LIN {X 0,Y 474.607,Z 153.704,A -85,B 0,C 180,E1 -7123.223,E2 -7123.223} C_VEL
LIN {X 0,Y 474.574,Z 152.961,A -85,B 0,C 180,E1 -7123.313,E2 -7123.313} C_VEL
LIN {X 0,Y 474.891,Z 139.856,A -85,B 0,C 180,E1 -7126.331,E2 -7126.331} C_VEL
LIN {X 0,Y 475.169,Z 128.62,A -85,B 0,C 180,E1 -7128.989,E2 -7128.989} C_VEL
LIN {X 0,Y 474.717,Z 124.266,A -85,B 0,C 180,E1 -7130.105,E2 -7130.105} C_VEL
LIN {X 0,Y 474.611,Z 124.173,A -85,B 0,C 180,E1 -7133.566,E2 -7133.566} C_VEL
LIN {X 0,Y 474.655,Z 124.176,A -85,B 0,C 180,E1 -7136.372,E2 -7136.372} C_VEL
LIN {X 0,Y 474.621,Z 124.172,A -85,B 0,C 180,E1 -7139.252,E2 -7139.252} C_VEL
LIN {X 0,Y 474.614,Z 124.178,A -85,B 0,C 180,E1 -7142.43,E2 -7142.43} C_VEL
LIN {X 0,Y 474.617,Z 124.174,A -85,B 0,C 180,E1 -7145.469,E2 -7145.469} C_VEL
LIN {X 0,Y 474.611,Z 124.175,A -85,B 0,C 180,E1 -7148.457,E2 -7148.457} C_VEL
LIN {X 0,Y 474.627,Z 124.172,A -85,B 0,C 180,E1 -7150.959,E2 -7150.959} C_VEL
LIN {X 0,Y 474.605,Z 124.177,A -85,B 0,C 180,E1 -7154.105,E2 -7154.105} C_VEL
LIN {X 0,Y 474.613,Z 124.175,A -85,B 0,C 180,E1 -7157.065,E2 -7157.065} C_VEL
LIN {X 0,Y 474.617,Z 124.173,A -85,B 0,C 180,E1 -7160.354,E2 -7160.354} C_VEL
LIN {X 0,Y 474.591,Z 124.18,A -85,B 0,C 180,E1 -7163.677,E2 -7163.677} C_VEL
LIN {X 0,Y 474.642,Z 124.172,A -85,B 0,C 180,E1 -7166.78,E2 -7166.78} C_VEL
LIN {X 0,Y 474.604,Z 124.175,A -85,B 0,C 180,E1 -7169.77,E2 -7169.77} C_VEL
LIN {X 0,Y 474.696,Z 124.167,A -85,B 0,C 180,E1 -7172.68,E2 -7172.68} C_VEL
LIN {X 0,Y 474.656,Z 124.169,A -85,B 0,C 180,E1 -7175.507,E2 -7175.507} C_VEL
LIN {X 0,Y 474.67,Z 124.169,A -85,B 0,C 180,E1 -7179.185,E2 -7179.185} C_VEL
LIN {X 0,Y 474.656,Z 124.168,A -85,B 0,C 180,E1 -7181.884,E2 -7181.884} C_VEL
LIN {X 0,Y 474.699,Z 124.171,A -85,B 0,C 180,E1 -7184.544,E2 -7184.544} C_VEL
LIN {X 0,Y 474.738,Z 124.161,A -85,B 0,C 180,E1 -7188.038,E2 -7188.038} C_VEL
LIN {X 0,Y 474.727,Z 124.159,A -85,B 0,C 180,E1 -7191.486,E2 -7191.486} C_VEL
LIN {X 0,Y 474.778,Z 124.159,A -85,B 0,C 180,E1 -7194.052,E2 -7194.052} C_VEL
LIN {X 0,Y 474.893,Z 124.14,A -85,B 0,C 180,E1 -7197.455,E2 -7197.455} C_VEL
LIN {X 0,Y 474.911,Z 124.144,A -85,B 0,C 180,E1 -7200,E2 -7200} C_VEL
LIN {X 0,Y 474.893,Z 124.139,A -85,B 0,C 180,E1 -7202.545,E2 -7202.545} C_VEL
LIN {X 0,Y 474.777,Z 124.158,A -85,B 0,C 180,E1 -7205.948,E2 -7205.948} C_VEL
LIN {X 0,Y 474.726,Z 124.159,A -85,B 0,C 180,E1 -7208.513,E2 -7208.513} C_VEL
LIN {X 0,Y 474.703,Z 124.165,A -85,B 0,C 180,E1 -7211.962,E2 -7211.962} C_VEL
LIN {X 0,Y 474.698,Z 124.17,A -85,B 0,C 180,E1 -7215.456,E2 -7215.456} C_VEL
LIN {X 0,Y 474.664,Z 124.172,A -85,B 0,C 180,E1 -7219.01,E2 -7219.01} C_VEL
LIN {X 0,Y 474.586,Z 124.178,A -85,B 0,C 180,E1 -7221.729,E2 -7221.729} C_VEL
LIN {X 0,Y 474.655,Z 124.17,A -85,B 0,C 180,E1 -7224.493,E2 -7224.493} C_VEL
LIN {X 0,Y 474.679,Z 124.168,A -85,B 0,C 180,E1 -7227.334,E2 -7227.334} C_VEL
LIN {X 0,Y 474.603,Z 124.176,A -85,B 0,C 180,E1 -7230.23,E2 -7230.23} C_VEL
LIN {X 0,Y 474.641,Z 124.172,A -85,B 0,C 180,E1 -7233.22,E2 -7233.22} C_VEL
LIN {X 0,Y 474.59,Z 124.181,A -85,B 0,C 180,E1 -7236.323,E2 -7236.323} C_VEL
LIN {X 0,Y 474.616,Z 124.173,A -85,B 0,C 180,E1 -7239.646,E2 -7239.646} C_VEL
LIN {X 0,Y 474.613,Z 124.175,A -85,B 0,C 180,E1 -7242.934,E2 -7242.934} C_VEL
LIN {X 0,Y 474.604,Z 124.178,A -85,B 0,C 180,E1 -7245.895,E2 -7245.895} C_VEL
LIN {X 0,Y 474.626,Z 124.172,A -85,B 0,C 180,E1 -7249.041,E2 -7249.041} C_VEL
LIN {X 0,Y 474.609,Z 124.178,A -85,B 0,C 180,E1 -7251.704,E2 -7251.704} C_VEL
LIN {X 0,Y 474.626,Z 124.172,A -85,B 0,C 180,E1 -7254.726,E2 -7254.726} C_VEL
LIN {X 0,Y 474.634,Z 124.179,A -85,B 0,C 180,E1 -7257.788,E2 -7257.788} C_VEL
LIN {X 0,Y 474.623,Z 124.173,A -85,B 0,C 180,E1 -7260.885,E2 -7260.885} C_VEL
LIN {X 0,Y 474.661,Z 124.175,A -85,B 0,C 180,E1 -7263.629,E2 -7263.629} C_VEL
LIN {X 0,Y 474.635,Z 124.143,A -85,B 0,C 180,E1 -7266.642,E2 -7266.642} C_VEL
LIN {X 0,Y 474.654,Z 124.24,A -85,B 0,C 180,E1 -7267.156,E2 -7267.156} C_VEL
LIN {X 0,Y 475.653,Z 130.342,A -85,B 0,C 180,E1 -7268.568,E2 -7268.568} C_VEL
LIN {X 0,Y 475.455,Z 140.784,A -85,B 0,C 180,E1 -7270.799,E2 -7270.799} C_VEL
LIN {X 0,Y 474.832,Z 156.822,A -85,B 0,C 180,E1 -7274.168,E2 -7274.168} C_VEL
LIN {X 0,Y 474.475,Z 169.531,A -85,B 0,C 180,E1 -7276.78,E2 -7276.78} C_VEL
LIN {X 0,Y 474.997,Z 173.212,A -85,B 0,C 180,E1 -7276.9,E2 -7276.9} C_VEL
LIN {X 0,Y 476.416,Z 185.772,A -85,B 0,C 180,E1 -7277.13,E2 -7277.13} C_VEL
LIN {X 0,Y 476.155,Z 245.998,A -85,B 0,C 180,E1 -7278.055,E2 -7278.055} C_VEL
LIN {X 0,Y 475.911,Z 254.89,A -85,B 0,C 180,E1 -7278.285,E2 -7278.285} C_VEL
LIN {X 0,Y 475.705,Z 264.57,A -85,B 0,C 180,E1 -7278.658,E2 -7278.658} C_VEL
LIN {X 0,Y 475.452,Z 273.742,A -85,B 0,C 180,E1 -7279.137,E2 -7279.137} C_VEL
LIN {X 0,Y 475.067,Z 284.557,A -85,B 0,C 180,E1 -7279.882,E2 -7279.882} C_VEL
LIN {X 0,Y 474.683,Z 293.871,A -85,B 0,C 180,E1 -7280.735,E2 -7280.735} C_VEL
LIN {X 0,Y 474.468,Z 300.546,A -85,B 0,C 180,E1 -7281.482,E2 -7281.482} C_VEL
LIN {X 0,Y 474.248,Z 306.882,A -85,B 0,C 180,E1 -7282.336,E2 -7282.336} C_VEL
LIN {X 0,Y 474.068,Z 312.147,A -85,B 0,C 180,E1 -7283.189,E2 -7283.189} C_VEL
LIN {X 0,Y 473.99,Z 316.538,A -85,B 0,C 180,E1 -7284.043,E2 -7284.043} C_VEL
LIN {X 0,Y 473.795,Z 321.713,A -85,B 0,C 180,E1 -7285.321,E2 -7285.321} C_VEL
LIN {X 0,Y 473.826,Z 325.514,A -85,B 0,C 180,E1 -7286.599,E2 -7286.599} C_VEL
LIN {X 0,Y 473.727,Z 327.26,A -85,B 0,C 180,E1 -7287.449,E2 -7287.449} C_VEL
LIN {X 0,Y 473.693,Z 328.512,A -85,B 0,C 180,E1 -7288.3,E2 -7288.3} C_VEL
LIN {X 0,Y 473.686,Z 329.292,A -85,B 0,C 180,E1 -7289.15,E2 -7289.15} C_VEL
LIN {X 0,Y 473.668,Z 329.587,A -85,B 0,C 180,E1 -7290,E2 -7290} C_VEL
LIN {X 0,Y 473.686,Z 329.291,A -85,B 0,C 180,E1 -7290.85,E2 -7290.85} C_VEL
LIN {X 0,Y 473.693,Z 328.509,A -85,B 0,C 180,E1 -7291.701,E2 -7291.701} C_VEL
LIN {X 0,Y 473.727,Z 327.256,A -85,B 0,C 180,E1 -7292.551,E2 -7292.551} C_VEL
LIN {X 0,Y 473.82,Z 324.353,A -85,B 0,C 180,E1 -7293.827,E2 -7293.827} C_VEL
LIN {X 0,Y 473.795,Z 321.706,A -85,B 0,C 180,E1 -7294.68,E2 -7294.68} C_VEL
LIN {X 0,Y 473.987,Z 316.527,A -85,B 0,C 180,E1 -7295.958,E2 -7295.958} C_VEL
LIN {X 0,Y 474.123,Z 309.701,A -85,B 0,C 180,E1 -7297.239,E2 -7297.239} C_VEL
LIN {X 0,Y 474.398,Z 302.239,A -85,B 0,C 180,E1 -7298.305,E2 -7298.305} C_VEL
LIN {X 0,Y 474.668,Z 294.88,A -85,B 0,C 180,E1 -7299.159,E2 -7299.159} C_VEL
LIN {X 0,Y 474.993,Z 287.001,A -85,B 0,C 180,E1 -7299.905,E2 -7299.905} C_VEL
LIN {X 0,Y 475.285,Z 278.674,A -85,B 0,C 180,E1 -7300.544,E2 -7300.544} C_VEL
LIN {X 0,Y 475.615,Z 268.044,A -85,B 0,C 180,E1 -7301.183,E2 -7301.183} C_VEL
LIN {X 0,Y 475.856,Z 256.486,A -85,B 0,C 180,E1 -7301.663,E2 -7301.663} C_VEL
LIN {X 0,Y 476.109,Z 246.824,A -85,B 0,C 180,E1 -7301.927,E2 -7301.927} C_VEL
LIN {X 0,Y 476.329,Z 197.947,A -85,B 0,C 180,E1 -7302.686,E2 -7302.686} C_VEL
LIN {X 0,Y 476.185,Z 182.261,A -85,B 0,C 180,E1 -7302.928,E2 -7302.928} C_VEL
LIN {X 0,Y 474.503,Z 169.838,A -85,B 0,C 180,E1 -7303.189,E2 -7303.189} C_VEL
LIN {X 0,Y 474.633,Z 164.918,A -85,B 0,C 180,E1 -7304.142,E2 -7304.142} C_VEL
LIN {X 0,Y 475.093,Z 149.174,A -85,B 0,C 180,E1 -7307.431,E2 -7307.431} C_VEL
LIN {X 0,Y 475.598,Z 135.504,A -85,B 0,C 180,E1 -7310.32,E2 -7310.32} C_VEL
LIN {X 0,Y 475.533,Z 129.184,A -85,B 0,C 180,E1 -7311.684,E2 -7311.684} C_VEL
LIN {X 0,Y 474.653,Z 124.232,A -85,B 0,C 180,E1 -7312.844,E2 -7312.844} C_VEL
LIN {X 0,Y 474.671,Z 124.167,A -85,B 0,C 180,E1 -7315.428,E2 -7315.428} C_VEL
LIN {X 0,Y 474.646,Z 124.176,A -85,B 0,C 180,E1 -7318.283,E2 -7318.283} C_VEL
LIN {X 0,Y 474.599,Z 124.175,A -85,B 0,C 180,E1 -7321.218,E2 -7321.218} C_VEL
LIN {X 0,Y 474.633,Z 124.178,A -85,B 0,C 180,E1 -7324.241,E2 -7324.241} C_VEL
LIN {X 0,Y 474.59,Z 124.177,A -85,B 0,C 180,E1 -7327.384,E2 -7327.384} C_VEL
LIN {X 0,Y 474.628,Z 124.175,A -85,B 0,C 180,E1 -7329.648,E2 -7329.648} C_VEL
LIN {X 0,Y 474.607,Z 124.174,A -85,B 0,C 180,E1 -7332.935,E2 -7332.935} C_VEL
LIN {X 0,Y 474.605,Z 124.18,A -85,B 0,C 180,E1 -7335.895,E2 -7335.895} C_VEL
LIN {X 0,Y 474.628,Z 124.173,A -85,B 0,C 180,E1 -7339.041,E2 -7339.041} C_VEL
LIN {X 0,Y 474.611,Z 124.179,A -85,B 0,C 180,E1 -7341.704,E2 -7341.704} C_VEL
LIN {X 0,Y 474.63,Z 124.172,A -85,B 0,C 180,E1 -7344.726,E2 -7344.726} C_VEL
LIN {X 0,Y 474.636,Z 124.172,A -85,B 0,C 180,E1 -7347.788,E2 -7347.788} C_VEL
LIN {X 0,Y 474.625,Z 124.176,A -85,B 0,C 180,E1 -7350.885,E2 -7350.885} C_VEL
LIN {X 0,Y 474.661,Z 124.169,A -85,B 0,C 180,E1 -7353.629,E2 -7353.629} C_VEL
LIN {X 0,Y 474.637,Z 124.174,A -85,B 0,C 180,E1 -7356.642,E2 -7356.642} C_VEL
LIN {X 0,Y 474.656,Z 124.168,A -85,B 0,C 180,E1 -7360.09,E2 -7360.09} C_VEL
LIN {X 0,Y 474.652,Z 124.176,A -85,B 0,C 180,E1 -7362.775,E2 -7362.775} C_VEL
LIN {X 0,Y 474.649,Z 124.169,A -85,B 0,C 180,E1 -7365.421,E2 -7365.421} C_VEL
LIN {X 0,Y 474.706,Z 124.164,A -85,B 0,C 180,E1 -7368.038,E2 -7368.038} C_VEL
LIN {X 0,Y 474.729,Z 124.159,A -85,B 0,C 180,E1 -7371.487,E2 -7371.487} C_VEL
LIN {X 0,Y 474.774,Z 124.158,A -85,B 0,C 180,E1 -7374.052,E2 -7374.052} C_VEL
LIN {X 0,Y 474.895,Z 124.139,A -85,B 0,C 180,E1 -7377.455,E2 -7377.455} C_VEL
LIN {X 0,Y 474.913,Z 124.143,A -85,B 0,C 180,E1 -7380,E2 -7380} C_VEL
LIN {X 0,Y 474.895,Z 124.14,A -85,B 0,C 180,E1 -7382.545,E2 -7382.545} C_VEL
LIN {X 0,Y 474.78,Z 124.159,A -85,B 0,C 180,E1 -7385.948,E2 -7385.948} C_VEL
LIN {X 0,Y 474.73,Z 124.159,A -85,B 0,C 180,E1 -7388.514,E2 -7388.514} C_VEL
LIN {X 0,Y 474.741,Z 124.161,A -85,B 0,C 180,E1 -7391.962,E2 -7391.962} C_VEL
LIN {X 0,Y 474.683,Z 124.169,A -85,B 0,C 180,E1 -7395.768,E2 -7395.768} C_VEL
LIN {X 0,Y 474.666,Z 124.17,A -85,B 0,C 180,E1 -7399.01,E2 -7399.01} C_VEL
LIN {X 0,Y 474.59,Z 124.178,A -85,B 0,C 180,E1 -7401.729,E2 -7401.729} C_VEL
LIN {X 0,Y 474.656,Z 124.169,A -85,B 0,C 180,E1 -7404.493,E2 -7404.493} C_VEL
LIN {X 0,Y 474.683,Z 124.169,A -85,B 0,C 180,E1 -7407.334,E2 -7407.334} C_VEL
LIN {X 0,Y 474.607,Z 124.175,A -85,B 0,C 180,E1 -7410.23,E2 -7410.23} C_VEL
LIN {X 0,Y 474.644,Z 124.172,A -85,B 0,C 180,E1 -7413.22,E2 -7413.22} C_VEL
LIN {X 0,Y 474.594,Z 124.179,A -85,B 0,C 180,E1 -7416.323,E2 -7416.323} C_VEL
LIN {X 0,Y 474.619,Z 124.172,A -85,B 0,C 180,E1 -7419.646,E2 -7419.646} C_VEL
LIN {X 0,Y 474.625,Z 124.176,A -85,B 0,C 180,E1 -7422.237,E2 -7422.237} C_VEL
LIN {X 0,Y 474.618,Z 124.173,A -85,B 0,C 180,E1 -7425.298,E2 -7425.298} C_VEL
LIN {X 0,Y 474.622,Z 124.18,A -85,B 0,C 180,E1 -7428.215,E2 -7428.215} C_VEL
LIN {X 0,Y 474.646,Z 124.173,A -85,B 0,C 180,E1 -7430.454,E2 -7430.454} C_VEL
LIN {X 0,Y 474.594,Z 124.179,A -85,B 0,C 180,E1 -7433.677,E2 -7433.677} C_VEL
LIN {X 0,Y 474.635,Z 124.171,A -85,B 0,C 180,E1 -7436.779,E2 -7436.779} C_VEL
LIN {X 0,Y 474.608,Z 124.181,A -85,B 0,C 180,E1 -7439.77,E2 -7439.77} C_VEL
LIN {X 0,Y 474.699,Z 124.162,A -85,B 0,C 180,E1 -7442.68,E2 -7442.68} C_VEL
LIN {X 0,Y 474.643,Z 124.176,A -85,B 0,C 180,E1 -7445.506,E2 -7445.506} C_VEL
LIN {X 0,Y 474.678,Z 124.172,A -85,B 0,C 180,E1 -7449.186,E2 -7449.186} C_VEL
LIN {X 0,Y 474.748,Z 124.342,A -85,B 0,C 180,E1 -7450.037,E2 -7450.037} C_VEL
LIN {X 0,Y 474.933,Z 125.674,A -85,B 0,C 180,E1 -7450.378,E2 -7450.378} C_VEL
LIN {X 0,Y 474.496,Z 128.362,A -85,B 0,C 180,E1 -7451.009,E2 -7451.009} C_VEL
LIN {X 0,Y 471.684,Z 133.031,A -85,B 0,C 180,E1 -7452.012,E2 -7452.012} C_VEL
LIN {X 0,Y 468.637,Z 137.768,A -85,B 0,C 180,E1 -7453.024,E2 -7453.024} C_VEL
LIN {X 0,Y 467.867,Z 140.57,A -85,B 0,C 180,E1 -7453.662,E2 -7453.662} C_VEL
LIN {X 0,Y 467.56,Z 153.292,A -85,B 0,C 180,E1 -7456.617,E2 -7456.617} C_VEL
LIN {X 0,Y 467.786,Z 155.144,A -85,B 0,C 180,E1 -7456.72,E2 -7456.72} C_VEL
LIN {X 0,Y 469.597,Z 167.722,A -85,B 0,C 180,E1 -7456.966,E2 -7456.966} C_VEL
LIN {X 0,Y 469.251,Z 229.25,A -85,B 0,C 180,E1 -7457.924,E2 -7457.924} C_VEL
LIN {X 0,Y 469.09,Z 238.375,A -85,B 0,C 180,E1 -7458.166,E2 -7458.166} C_VEL
LIN {X 0,Y 468.894,Z 247.98,A -85,B 0,C 180,E1 -7458.545,E2 -7458.545} C_VEL
LIN {X 0,Y 468.654,Z 256.16,A -85,B 0,C 180,E1 -7458.977,E2 -7458.977} C_VEL
LIN {X 0,Y 468.325,Z 265.766,A -85,B 0,C 180,E1 -7459.625,E2 -7459.625} C_VEL
LIN {X 0,Y 467.982,Z 275.586,A -85,B 0,C 180,E1 -7460.491,E2 -7460.491} C_VEL
LIN {X 0,Y 467.625,Z 283.328,A -85,B 0,C 180,E1 -7461.356,E2 -7461.356} C_VEL
LIN {X 0,Y 467.337,Z 289.691,A -85,B 0,C 180,E1 -7462.221,E2 -7462.221} C_VEL
LIN {X 0,Y 467.207,Z 295.186,A -85,B 0,C 180,E1 -7463.126,E2 -7463.126} C_VEL
LIN {X 0,Y 467.083,Z 299.395,A -85,B 0,C 180,E1 -7463.954,E2 -7463.954} C_VEL
LIN {X 0,Y 466.82,Z 304.587,A -85,B 0,C 180,E1 -7465.25,E2 -7465.25} C_VEL
LIN {X 0,Y 466.846,Z 307.253,A -85,B 0,C 180,E1 -7466.115,E2 -7466.115} C_VEL
LIN {X 0,Y 466.675,Z 310.175,A -85,B 0,C 180,E1 -7467.41,E2 -7467.41} C_VEL
LIN {X 0,Y 466.608,Z 311.455,A -85,B 0,C 180,E1 -7468.274,E2 -7468.274} C_VEL
LIN {X 0,Y 466.589,Z 312.264,A -85,B 0,C 180,E1 -7469.137,E2 -7469.137} C_VEL
LIN {X 0,Y 466.599,Z 312.572,A -85,B 0,C 180,E1 -7470,E2 -7470} C_VEL
LIN {X 0,Y 466.589,Z 312.299,A -85,B 0,C 180,E1 -7470.863,E2 -7470.863} C_VEL
LIN {X 0,Y 466.608,Z 311.558,A -85,B 0,C 180,E1 -7471.726,E2 -7471.726} C_VEL
LIN {X 0,Y 466.674,Z 310.348,A -85,B 0,C 180,E1 -7472.589,E2 -7472.589} C_VEL
LIN {X 0,Y 466.835,Z 307.5,A -85,B 0,C 180,E1 -7473.884,E2 -7473.884} C_VEL
LIN {X 0,Y 466.814,Z 304.911,A -85,B 0,C 180,E1 -7474.75,E2 -7474.75} C_VEL
LIN {X 0,Y 467.065,Z 299.805,A -85,B 0,C 180,E1 -7476.046,E2 -7476.046} C_VEL
LIN {X 0,Y 467.203,Z 294.315,A -85,B 0,C 180,E1 -7477.129,E2 -7477.129} C_VEL
LIN {X 0,Y 467.459,Z 287.422,A -85,B 0,C 180,E1 -7478.211,E2 -7478.211} C_VEL
LIN {X 0,Y 467.78,Z 279.505,A -85,B 0,C 180,E1 -7479.185,E2 -7479.185} C_VEL
LIN {X 0,Y 468.107,Z 271.953,A -85,B 0,C 180,E1 -7479.942,E2 -7479.942} C_VEL
LIN {X 0,Y 468.374,Z 264.042,A -85,B 0,C 180,E1 -7480.592,E2 -7480.592} C_VEL
LIN {X 0,Y 468.713,Z 255.875,A -85,B 0,C 180,E1 -7481.131,E2 -7481.131} C_VEL
LIN {X 0,Y 468.89,Z 247.61,A -85,B 0,C 180,E1 -7481.564,E2 -7481.564} C_VEL
LIN {X 0,Y 469.144,Z 238.696,A -85,B 0,C 180,E1 -7481.914,E2 -7481.914} C_VEL
LIN {X 0,Y 469.301,Z 229.511,A -85,B 0,C 180,E1 -7482.162,E2 -7482.162} C_VEL
LIN {X 0,Y 469.537,Z 166.026,A -85,B 0,C 180,E1 -7483.155,E2 -7483.155} C_VEL
LIN {X 0,Y 467.588,Z 153.818,A -85,B 0,C 180,E1 -7483.425,E2 -7483.425} C_VEL
LIN {X 0,Y 467.568,Z 153.07,A -85,B 0,C 180,E1 -7483.517,E2 -7483.517} C_VEL
LIN {X 0,Y 467.892,Z 139.938,A -85,B 0,C 180,E1 -7486.582,E2 -7486.582} C_VEL
LIN {X 0,Y 468.18,Z 129.978,A -85,B 0,C 180,E1 -7488.966,E2 -7488.966} C_VEL
LIN {X 0,Y 467.681,Z 125.139,A -85,B 0,C 180,E1 -7490.22,E2 -7490.22} C_VEL
LIN {X 0,Y 467.563,Z 125.054,A -85,B 0,C 180,E1 -7493.943,E2 -7493.943} C_VEL
LIN {X 0,Y 467.614,Z 125.048,A -85,B 0,C 180,E1 -7496.8,E2 -7496.8} C_VEL
LIN {X 0,Y 467.554,Z 125.054,A -85,B 0,C 180,E1 -7499.738,E2 -7499.738} C_VEL
LIN {X 0,Y 467.581,Z 125.051,A -85,B 0,C 180,E1 -7502.758,E2 -7502.758} C_VEL
LIN {X 0,Y 467.555,Z 125.058,A -85,B 0,C 180,E1 -7505.889,E2 -7505.889} C_VEL
LIN {X 0,Y 467.582,Z 125.05,A -85,B 0,C 180,E1 -7509.144,E2 -7509.144} C_VEL
LIN {X 0,Y 467.586,Z 125.049,A -85,B 0,C 180,E1 -7512.567,E2 -7512.567} C_VEL
LIN {X 0,Y 467.565,Z 125.052,A -85,B 0,C 180,E1 -7515.052,E2 -7515.052} C_VEL
LIN {X 0,Y 467.588,Z 125.054,A -85,B 0,C 180,E1 -7517.44,E2 -7517.44} C_VEL
LIN {X 0,Y 467.559,Z 125.053,A -85,B 0,C 180,E1 -7520.853,E2 -7520.853} C_VEL
LIN {X 0,Y 467.561,Z 125.052,A -85,B 0,C 180,E1 -7524.26,E2 -7524.26} C_VEL
LIN {X 0,Y 467.581,Z 125.056,A -85,B 0,C 180,E1 -7527.321,E2 -7527.321} C_VEL
LIN {X 0,Y 467.569,Z 125.053,A -85,B 0,C 180,E1 -7530.667,E2 -7530.667} C_VEL
LIN {X 0,Y 467.615,Z 125.05,A -85,B 0,C 180,E1 -7533.2,E2 -7533.2} C_VEL
LIN {X 0,Y 467.591,Z 125.051,A -85,B 0,C 180,E1 -7536.468,E2 -7536.468} C_VEL
LIN {X 0,Y 467.623,Z 125.044,A -85,B 0,C 180,E1 -7539.777,E2 -7539.777} C_VEL
LIN {X 0,Y 467.608,Z 125.052,A -85,B 0,C 180,E1 -7542.507,E2 -7542.507} C_VEL
LIN {X 0,Y 467.605,Z 125.047,A -85,B 0,C 180,E1 -7545.196,E2 -7545.196} C_VEL
LIN {X 0,Y 467.682,Z 125.038,A -85,B 0,C 180,E1 -7547.855,E2 -7547.855} C_VEL
LIN {X 0,Y 467.68,Z 125.037,A -85,B 0,C 180,E1 -7551.357,E2 -7551.357} C_VEL
LIN {X 0,Y 467.742,Z 125.034,A -85,B 0,C 180,E1 -7553.963,E2 -7553.963} C_VEL
LIN {X 0,Y 467.858,Z 125.016,A -85,B 0,C 180,E1 -7557.417,E2 -7557.417} C_VEL
LIN {X 0,Y 467.882,Z 125.02,A -85,B 0,C 180,E1 -7560,E2 -7560} C_VEL
LIN {X 0,Y 467.858,Z 125.015,A -85,B 0,C 180,E1 -7562.583,E2 -7562.583} C_VEL
LIN {X 0,Y 467.742,Z 125.033,A -85,B 0,C 180,E1 -7566.037,E2 -7566.037} C_VEL
LIN {X 0,Y 467.68,Z 125.037,A -85,B 0,C 180,E1 -7568.643,E2 -7568.643} C_VEL
LIN {X 0,Y 467.654,Z 125.041,A -85,B 0,C 180,E1 -7572.145,E2 -7572.145} C_VEL
LIN {X 0,Y 467.638,Z 125.046,A -85,B 0,C 180,E1 -7575.695,E2 -7575.695} C_VEL
LIN {X 0,Y 467.616,Z 125.047,A -85,B 0,C 180,E1 -7578.765,E2 -7578.765} C_VEL
LIN {X 0,Y 467.579,Z 125.056,A -85,B 0,C 180,E1 -7581.268,E2 -7581.268} C_VEL
LIN {X 0,Y 467.57,Z 125.051,A -85,B 0,C 180,E1 -7583.943,E2 -7583.943} C_VEL
LIN {X 0,Y 467.615,Z 125.051,A -85,B 0,C 180,E1 -7586.8,E2 -7586.8} C_VEL
LIN {X 0,Y 467.552,Z 125.053,A -85,B 0,C 180,E1 -7589.738,E2 -7589.738} C_VEL
LIN {X 0,Y 467.581,Z 125.057,A -85,B 0,C 180,E1 -7592.758,E2 -7592.758} C_VEL
LIN {X 0,Y 467.554,Z 125.053,A -85,B 0,C 180,E1 -7595.889,E2 -7595.889} C_VEL
LIN {X 0,Y 467.558,Z 125.053,A -85,B 0,C 180,E1 -7599.147,E2 -7599.147} C_VEL
LIN {X 0,Y 467.585,Z 125.054,A -85,B 0,C 180,E1 -7602.567,E2 -7602.567} C_VEL
LIN {X 0,Y 467.564,Z 125.052,A -85,B 0,C 180,E1 -7605.053,E2 -7605.053} C_VEL
LIN {X 0,Y 467.587,Z 125.049,A -85,B 0,C 180,E1 -7607.44,E2 -7607.44} C_VEL
LIN {X 0,Y 467.58,Z 125.05,A -85,B 0,C 180,E1 -7610.855,E2 -7610.855} C_VEL
LIN {X 0,Y 467.56,Z 125.055,A -85,B 0,C 180,E1 -7614.261,E2 -7614.261} C_VEL
LIN {X 0,Y 467.579,Z 125.052,A -85,B 0,C 180,E1 -7617.321,E2 -7617.321} C_VEL
LIN {X 0,Y 467.569,Z 125.051,A -85,B 0,C 180,E1 -7620.668,E2 -7620.668} C_VEL
LIN {X 0,Y 467.616,Z 125.048,A -85,B 0,C 180,E1 -7623.2,E2 -7623.2} C_VEL
LIN {X 0,Y 467.592,Z 125.02,A -85,B 0,C 180,E1 -7626.469,E2 -7626.469} C_VEL
LIN {X 0,Y 467.604,Z 125.087,A -85,B 0,C 180,E1 -7626.998,E2 -7626.998} C_VEL
LIN {X 0,Y 468.321,Z 129.066,A -85,B 0,C 180,E1 -7627.965,E2 -7627.965} C_VEL
LIN {X 0,Y 468.681,Z 134.347,A -85,B 0,C 180,E1 -7629.137,E2 -7629.137} C_VEL
LIN {X 0,Y 468.193,Z 146.966,A -85,B 0,C 180,E1 -7631.852,E2 -7631.852} C_VEL
LIN {X 0,Y 467.728,Z 161.661,A -85,B 0,C 180,E1 -7634.978,E2 -7634.978} C_VEL
LIN {X 0,Y 467.46,Z 169.471,A -85,B 0,C 180,E1 -7636.585,E2 -7636.585} C_VEL
LIN {X 0,Y 467.959,Z 173.317,A -85,B 0,C 180,E1 -7636.703,E2 -7636.703} C_VEL
LIN {X 0,Y 469.51,Z 185.877,A -85,B 0,C 180,E1 -7636.941,E2 -7636.941} C_VEL
LIN {X 0,Y 469.217,Z 245.925,A -85,B 0,C 180,E1 -7637.877,E2 -7637.877} C_VEL
LIN {X 0,Y 468.946,Z 255.601,A -85,B 0,C 180,E1 -7638.136,E2 -7638.136} C_VEL
LIN {X 0,Y 468.685,Z 265.657,A -85,B 0,C 180,E1 -7638.54,E2 -7638.54} C_VEL
LIN {X 0,Y 468.383,Z 277.077,A -85,B 0,C 180,E1 -7639.19,E2 -7639.19} C_VEL
LIN {X 0,Y 468.034,Z 285.666,A -85,B 0,C 180,E1 -7639.838,E2 -7639.838} C_VEL
LIN {X 0,Y 467.647,Z 293.744,A -85,B 0,C 180,E1 -7640.594,E2 -7640.594} C_VEL
LIN {X 0,Y 467.426,Z 300.419,A -85,B 0,C 180,E1 -7641.353,E2 -7641.353} C_VEL
LIN {X 0,Y 467.207,Z 306.755,A -85,B 0,C 180,E1 -7642.219,E2 -7642.219} C_VEL
LIN {X 0,Y 467.002,Z 312.02,A -85,B 0,C 180,E1 -7643.085,E2 -7643.085} C_VEL
LIN {X 0,Y 466.897,Z 316.41,A -85,B 0,C 180,E1 -7643.952,E2 -7643.952} C_VEL
LIN {X 0,Y 466.721,Z 321.585,A -85,B 0,C 180,E1 -7645.25,E2 -7645.25} C_VEL
LIN {X 0,Y 466.724,Z 325.386,A -85,B 0,C 180,E1 -7646.547,E2 -7646.547} C_VEL
LIN {X 0,Y 466.65,Z 327.133,A -85,B 0,C 180,E1 -7647.411,E2 -7647.411} C_VEL
LIN {X 0,Y 466.603,Z 328.384,A -85,B 0,C 180,E1 -7648.274,E2 -7648.274} C_VEL
LIN {X 0,Y 466.587,Z 329.163,A -85,B 0,C 180,E1 -7649.137,E2 -7649.137} C_VEL
LIN {X 0,Y 466.597,Z 329.459,A -85,B 0,C 180,E1 -7650,E2 -7650} C_VEL
LIN {X 0,Y 466.587,Z 329.162,A -85,B 0,C 180,E1 -7650.863,E2 -7650.863} C_VEL
LIN {X 0,Y 466.603,Z 328.381,A -85,B 0,C 180,E1 -7651.726,E2 -7651.726} C_VEL
LIN {X 0,Y 466.65,Z 327.127,A -85,B 0,C 180,E1 -7652.59,E2 -7652.59} C_VEL
LIN {X 0,Y 466.711,Z 324.224,A -85,B 0,C 180,E1 -7653.886,E2 -7653.886} C_VEL
LIN {X 0,Y 466.721,Z 321.576,A -85,B 0,C 180,E1 -7654.751,E2 -7654.751} C_VEL
LIN {X 0,Y 466.892,Z 316.397,A -85,B 0,C 180,E1 -7656.049,E2 -7656.049} C_VEL
LIN {X 0,Y 467.05,Z 309.571,A -85,B 0,C 180,E1 -7657.349,E2 -7657.349} C_VEL
LIN {X 0,Y 467.355,Z 302.109,A -85,B 0,C 180,E1 -7658.431,E2 -7658.431} C_VEL
LIN {X 0,Y 467.631,Z 294.749,A -85,B 0,C 180,E1 -7659.298,E2 -7659.298} C_VEL
LIN {X 0,Y 467.99,Z 286.869,A -85,B 0,C 180,E1 -7660.054,E2 -7660.054} C_VEL
LIN {X 0,Y 468.279,Z 278.542,A -85,B 0,C 180,E1 -7660.704,E2 -7660.704} C_VEL
LIN {X 0,Y 468.651,Z 267.911,A -85,B 0,C 180,E1 -7661.352,E2 -7661.352} C_VEL
LIN {X 0,Y 468.915,Z 256.35,A -85,B 0,C 180,E1 -7661.838,E2 -7661.838} C_VEL
LIN {X 0,Y 469.168,Z 246.683,A -85,B 0,C 180,E1 -7662.106,E2 -7662.106} C_VEL
LIN {X 0,Y 469.49,Z 189.42,A -85,B 0,C 180,E1 -7663.003,E2 -7663.003} C_VEL
LIN {X 0,Y 469.193,Z 182.169,A -85,B 0,C 180,E1 -7663.123,E2 -7663.123} C_VEL
LIN {X 0,Y 467.494,Z 169.803,A -85,B 0,C 180,E1 -7663.383,E2 -7663.383} C_VEL
LIN {X 0,Y 467.516,Z 166.885,A -85,B 0,C 180,E1 -7663.918,E2 -7663.918} C_VEL
LIN {X 0,Y 467.995,Z 153.25,A -85,B 0,C 180,E1 -7666.803,E2 -7666.803} C_VEL
LIN {X 0,Y 468.569,Z 137.485,A -85,B 0,C 180,E1 -7670.18,E2 -7670.18} C_VEL
LIN {X 0,Y 468.625,Z 130.998,A -85,B 0,C 180,E1 -7671.594,E2 -7671.594} C_VEL
LIN {X 0,Y 467.659,Z 125.366,A -85,B 0,C 180,E1 -7672.883,E2 -7672.883} C_VEL
LIN {X 0,Y 467.596,Z 125.017,A -85,B 0,C 180,E1 -7673.267,E2 -7673.267} C_VEL
LIN {X 0,Y 467.611,Z 125.048,A -85,B 0,C 180,E1 -7675.84,E2 -7675.84} C_VEL
LIN {X 0,Y 467.577,Z 125.053,A -85,B 0,C 180,E1 -7678.75,E2 -7678.75} C_VEL
LIN {X 0,Y 467.583,Z 125.051,A -85,B 0,C 180,E1 -7681.74,E2 -7681.74} C_VEL
LIN {X 0,Y 467.565,Z 125.052,A -85,B 0,C 180,E1 -7684.833,E2 -7684.833} C_VEL
LIN {X 0,Y 467.565,Z 125.059,A -85,B 0,C 180,E1 -7688.045,E2 -7688.045} C_VEL
LIN {X 0,Y 467.578,Z 125.051,A -85,B 0,C 180,E1 -7691.277,E2 -7691.277} C_VEL
LIN {X 0,Y 467.55,Z 125.061,A -85,B 0,C 180,E1 -7693.82,E2 -7693.82} C_VEL
LIN {X 0,Y 467.551,Z 125.055,A -85,B 0,C 180,E1 -7696.255,E2 -7696.255} C_VEL
LIN {X 0,Y 467.579,Z 125.05,A -85,B 0,C 180,E1 -7698.723,E2 -7698.723} C_VEL
LIN {X 0,Y 467.566,Z 125.054,A -85,B 0,C 180,E1 -7701.956,E2 -7701.956} C_VEL
LIN {X 0,Y 467.569,Z 125.056,A -85,B 0,C 180,E1 -7705.168,E2 -7705.168} C_VEL
LIN {X 0,Y 467.584,Z 125.049,A -85,B 0,C 180,E1 -7708.26,E2 -7708.26} C_VEL
LIN {X 0,Y 467.578,Z 125.056,A -85,B 0,C 180,E1 -7711.251,E2 -7711.251} C_VEL
LIN {X 0,Y 467.611,Z 125.046,A -85,B 0,C 180,E1 -7714.16,E2 -7714.16} C_VEL
LIN {X 0,Y 467.578,Z 125.057,A -85,B 0,C 180,E1 -7716.996,E2 -7716.996} C_VEL
LIN {X 0,Y 467.624,Z 125.044,A -85,B 0,C 180,E1 -7719.777,E2 -7719.777} C_VEL
LIN {X 0,Y 467.611,Z 125.051,A -85,B 0,C 180,E1 -7722.507,E2 -7722.507} C_VEL
LIN {X 0,Y 467.608,Z 125.047,A -85,B 0,C 180,E1 -7725.197,E2 -7725.197} C_VEL
LIN {X 0,Y 467.657,Z 125.041,A -85,B 0,C 180,E1 -7727.855,E2 -7727.855} C_VEL
LIN {X 0,Y 467.683,Z 125.037,A -85,B 0,C 180,E1 -7731.357,E2 -7731.357} C_VEL
LIN {X 0,Y 467.738,Z 125.033,A -85,B 0,C 180,E1 -7733.963,E2 -7733.963} C_VEL
LIN {X 0,Y 467.86,Z 125.015,A -85,B 0,C 180,E1 -7737.417,E2 -7737.417} C_VEL
LIN {X 0,Y 467.884,Z 125.019,A -85,B 0,C 180,E1 -7740,E2 -7740} C_VEL
LIN {X 0,Y 467.86,Z 125.016,A -85,B 0,C 180,E1 -7742.583,E2 -7742.583} C_VEL
LIN {X 0,Y 467.745,Z 125.034,A -85,B 0,C 180,E1 -7746.037,E2 -7746.037} C_VEL
LIN {X 0,Y 467.683,Z 125.037,A -85,B 0,C 180,E1 -7748.643,E2 -7748.643} C_VEL
LIN {X 0,Y 467.685,Z 125.038,A -85,B 0,C 180,E1 -7752.145,E2 -7752.145} C_VEL
LIN {X 0,Y 467.651,Z 125.043,A -85,B 0,C 180,E1 -7755.885,E2 -7755.885} C_VEL
LIN {X 0,Y 467.625,Z 125.051,A -85,B 0,C 180,E1 -7759.308,E2 -7759.308} C_VEL
LIN {X 0,Y 467.536,Z 125.055,A -85,B 0,C 180,E1 -7762.074,E2 -7762.074} C_VEL
LIN {X 0,Y 467.603,Z 125.051,A -85,B 0,C 180,E1 -7764.887,E2 -7764.887} C_VEL
LIN {X 0,Y 467.622,Z 125.045,A -85,B 0,C 180,E1 -7767.769,E2 -7767.769} C_VEL
LIN {X 0,Y 467.57,Z 125.057,A -85,B 0,C 180,E1 -7771.045,E2 -7771.045} C_VEL
LIN {X 0,Y 467.591,Z 125.05,A -85,B 0,C 180,E1 -7774.242,E2 -7774.242} C_VEL
LIN {X 0,Y 467.551,Z 125.055,A -85,B 0,C 180,E1 -7777.187,E2 -7777.187} C_VEL
LIN {X 0,Y 467.576,Z 125.054,A -85,B 0,C 180,E1 -7780.265,E2 -7780.265} C_VEL
LIN {X 0,Y 467.588,Z 125.055,A -85,B 0,C 180,E1 -7782.567,E2 -7782.567} C_VEL
LIN {X 0,Y 467.567,Z 125.052,A -85,B 0,C 180,E1 -7785.053,E2 -7785.053} C_VEL
LIN {X 0,Y 467.591,Z 125.048,A -85,B 0,C 180,E1 -7787.44,E2 -7787.44} C_VEL
LIN {X 0,Y 467.584,Z 125.05,A -85,B 0,C 180,E1 -7790.855,E2 -7790.855} C_VEL
LIN {X 0,Y 467.563,Z 125.056,A -85,B 0,C 180,E1 -7794.261,E2 -7794.261} C_VEL
LIN {X 0,Y 467.582,Z 125.05,A -85,B 0,C 180,E1 -7797.321,E2 -7797.321} C_VEL
LIN {X 0,Y 467.572,Z 125.051,A -85,B 0,C 180,E1 -7800.667,E2 -7800.667} C_VEL
LIN {X 0,Y 467.615,Z 125.047,A -85,B 0,C 180,E1 -7803.199,E2 -7803.199} C_VEL
LIN {X 0,Y 467.593,Z 125.05,A -85,B 0,C 180,E1 -7806.469,E2 -7806.469} C_VEL
LIN {X 0,Y 467.713,Z 125.289,A -85,B 0,C 180,E1 -7809.953,E2 -7809.953} C_VEL
LIN {X 0,Y 468.181,Z 130.797,A -85,B 0,C 180,E1 -7811.327,E2 -7811.327} C_VEL
LIN {X 0,Y 467.867,Z 140.57,A -85,B 0,C 180,E1 -7813.662,E2 -7813.662} C_VEL
LIN {X 0,Y 467.138,Z 142.456,A -85,B 0,C 180,E1 -7814.082,E2 -7814.082} C_VEL
LIN {X 0,Y 461.291,Z 148.792,A -85,B 0,C 180,E1 -7815.365,E2 -7815.365} C_VEL
LIN {X 0,Y 460.595,Z 150.702,A -85,B 0,C 180,E1 -7815.792,E2 -7815.792} C_VEL
LIN {X 0,Y 460.561,Z 153.716,A -85,B 0,C 180,E1 -7816.442,E2 -7816.442} C_VEL
LIN {X 0,Y 461.109,Z 157.23,A -85,B 0,C 180,E1 -7816.554,E2 -7816.554} C_VEL
LIN {X 0,Y 462.71,Z 167.878,A -85,B 0,C 180,E1 -7816.769,E2 -7816.769} C_VEL
LIN {X 0,Y 462.329,Z 229.398,A -85,B 0,C 180,E1 -7817.74,E2 -7817.74} C_VEL
LIN {X 0,Y 462.159,Z 238.516,A -85,B 0,C 180,E1 -7817.986,E2 -7817.986} C_VEL
LIN {X 0,Y 461.951,Z 248.118,A -85,B 0,C 180,E1 -7818.37,E2 -7818.37} C_VEL
LIN {X 0,Y 461.683,Z 256.296,A -85,B 0,C 180,E1 -7818.808,E2 -7818.808} C_VEL
LIN {X 0,Y 461.35,Z 265.901,A -85,B 0,C 180,E1 -7819.467,E2 -7819.467} C_VEL
LIN {X 0,Y 460.982,Z 275.719,A -85,B 0,C 180,E1 -7820.346,E2 -7820.346} C_VEL
LIN {X 0,Y 460.599,Z 283.46,A -85,B 0,C 180,E1 -7821.223,E2 -7821.223} C_VEL
LIN {X 0,Y 460.296,Z 289.823,A -85,B 0,C 180,E1 -7822.101,E2 -7822.101} C_VEL
LIN {X 0,Y 460.131,Z 295.863,A -85,B 0,C 180,E1 -7823.123,E2 -7823.123} C_VEL
LIN {X 0,Y 460.028,Z 299.525,A -85,B 0,C 180,E1 -7823.861,E2 -7823.861} C_VEL
LIN {X 0,Y 459.74,Z 304.717,A -85,B 0,C 180,E1 -7825.177,E2 -7825.177} C_VEL
LIN {X 0,Y 459.758,Z 307.383,A -85,B 0,C 180,E1 -7826.055,E2 -7826.055} C_VEL
LIN {X 0,Y 459.601,Z 310.304,A -85,B 0,C 180,E1 -7827.37,E2 -7827.37} C_VEL
LIN {X 0,Y 459.521,Z 311.584,A -85,B 0,C 180,E1 -7828.247,E2 -7828.247} C_VEL
LIN {X 0,Y 459.494,Z 312.393,A -85,B 0,C 180,E1 -7829.123,E2 -7829.123} C_VEL
LIN {X 0,Y 459.501,Z 312.701,A -85,B 0,C 180,E1 -7830,E2 -7830} C_VEL
LIN {X 0,Y 459.494,Z 312.427,A -85,B 0,C 180,E1 -7830.876,E2 -7830.876} C_VEL
LIN {X 0,Y 459.521,Z 311.686,A -85,B 0,C 180,E1 -7831.753,E2 -7831.753} C_VEL
LIN {X 0,Y 459.6,Z 310.476,A -85,B 0,C 180,E1 -7832.629,E2 -7832.629} C_VEL
LIN {X 0,Y 459.747,Z 307.627,A -85,B 0,C 180,E1 -7833.944,E2 -7833.944} C_VEL
LIN {X 0,Y 459.734,Z 305.038,A -85,B 0,C 180,E1 -7834.823,E2 -7834.823} C_VEL
LIN {X 0,Y 460.013,Z 299.932,A -85,B 0,C 180,E1 -7836.139,E2 -7836.139} C_VEL
LIN {X 0,Y 460.154,Z 294.441,A -85,B 0,C 180,E1 -7837.238,E2 -7837.238} C_VEL
LIN {X 0,Y 460.445,Z 287.547,A -85,B 0,C 180,E1 -7838.337,E2 -7838.337} C_VEL
LIN {X 0,Y 460.766,Z 279.629,A -85,B 0,C 180,E1 -7839.326,E2 -7839.326} C_VEL
LIN {X 0,Y 461.093,Z 272.077,A -85,B 0,C 180,E1 -7840.095,E2 -7840.095} C_VEL
LIN {X 0,Y 461.404,Z 264.165,A -85,B 0,C 180,E1 -7840.754,E2 -7840.754} C_VEL
LIN {X 0,Y 461.751,Z 255.996,A -85,B 0,C 180,E1 -7841.301,E2 -7841.301} C_VEL
LIN {X 0,Y 461.958,Z 247.729,A -85,B 0,C 180,E1 -7841.74,E2 -7841.74} C_VEL
LIN {X 0,Y 462.213,Z 238.811,A -85,B 0,C 180,E1 -7842.095,E2 -7842.095} C_VEL
LIN {X 0,Y 462.387,Z 229.728,A -85,B 0,C 180,E1 -7842.344,E2 -7842.344} C_VEL
LIN {X 0,Y 462.641,Z 166.786,A -85,B 0,C 180,E1 -7843.344,E2 -7843.344} C_VEL
LIN {X 0,Y 460.591,Z 153.95,A -85,B 0,C 180,E1 -7843.632,E2 -7843.632} C_VEL
LIN {X 0,Y 460.546,Z 153.185,A -85,B 0,C 180,E1 -7843.725,E2 -7843.725} C_VEL
LIN {X 0,Y 460.918,Z 140.021,A -85,B 0,C 180,E1 -7846.84,E2 -7846.84} C_VEL
LIN {X 0,Y 461.158,Z 130.657,A -85,B 0,C 180,E1 -7849.113,E2 -7849.113} C_VEL
LIN {X 0,Y 460.628,Z 126.034,A -85,B 0,C 180,E1 -7850.31,E2 -7850.31} C_VEL
LIN {X 0,Y 460.532,Z 125.928,A -85,B 0,C 180,E1 -7853.703,E2 -7853.703} C_VEL
LIN {X 0,Y 460.557,Z 125.93,A -85,B 0,C 180,E1 -7856.265,E2 -7856.265} C_VEL
LIN {X 0,Y 460.54,Z 125.926,A -85,B 0,C 180,E1 -7859.231,E2 -7859.231} C_VEL
LIN {X 0,Y 460.53,Z 125.934,A -85,B 0,C 180,E1 -7862.284,E2 -7862.284} C_VEL
LIN {X 0,Y 460.512,Z 125.931,A -85,B 0,C 180,E1 -7865.445,E2 -7865.445} C_VEL
LIN {X 0,Y 460.544,Z 125.926,A -85,B 0,C 180,E1 -7868.897,E2 -7868.897} C_VEL
LIN {X 0,Y 460.522,Z 125.932,A -85,B 0,C 180,E1 -7872.181,E2 -7872.181} C_VEL
LIN {X 0,Y 460.513,Z 125.934,A -85,B 0,C 180,E1 -7875.411,E2 -7875.411} C_VEL
LIN {X 0,Y 460.531,Z 125.928,A -85,B 0,C 180,E1 -7878.397,E2 -7878.397} C_VEL
LIN {X 0,Y 460.518,Z 125.934,A -85,B 0,C 180,E1 -7881.266,E2 -7881.266} C_VEL
LIN {X 0,Y 460.512,Z 125.93,A -85,B 0,C 180,E1 -7884.554,E2 -7884.554} C_VEL
LIN {X 0,Y 460.53,Z 125.93,A -85,B 0,C 180,E1 -7887.715,E2 -7887.715} C_VEL
LIN {X 0,Y 460.539,Z 125.93,A -85,B 0,C 180,E1 -7890.769,E2 -7890.769} C_VEL
LIN {X 0,Y 460.562,Z 125.924,A -85,B 0,C 180,E1 -7893.735,E2 -7893.735} C_VEL
LIN {X 0,Y 460.544,Z 125.93,A -85,B 0,C 180,E1 -7896.624,E2 -7896.624} C_VEL
LIN {X 0,Y 460.551,Z 125.926,A -85,B 0,C 180,E1 -7899.453,E2 -7899.453} C_VEL
LIN {X 0,Y 460.558,Z 125.927,A -85,B 0,C 180,E1 -7902.23,E2 -7902.23} C_VEL
LIN {X 0,Y 460.564,Z 125.926,A -85,B 0,C 180,E1 -7904.965,E2 -7904.965} C_VEL
LIN {X 0,Y 460.628,Z 125.916,A -85,B 0,C 180,E1 -7907.666,E2 -7907.666} C_VEL
LIN {X 0,Y 460.627,Z 125.916,A -85,B 0,C 180,E1 -7911.224,E2 -7911.224} C_VEL
LIN {X 0,Y 460.709,Z 125.909,A -85,B 0,C 180,E1 -7913.87,E2 -7913.87} C_VEL
LIN {X 0,Y 460.823,Z 125.892,A -85,B 0,C 180,E1 -7917.378,E2 -7917.378} C_VEL
LIN {X 0,Y 460.852,Z 125.895,A -85,B 0,C 180,E1 -7920,E2 -7920} C_VEL
LIN {X 0,Y 460.799,Z 125.895,A -85,B 0,C 180,E1 -7922.622,E2 -7922.622} C_VEL
LIN {X 0,Y 460.708,Z 125.908,A -85,B 0,C 180,E1 -7926.13,E2 -7926.13} C_VEL
LIN {X 0,Y 460.627,Z 125.916,A -85,B 0,C 180,E1 -7928.776,E2 -7928.776} C_VEL
LIN {X 0,Y 460.612,Z 125.917,A -85,B 0,C 180,E1 -7932.445,E2 -7932.445} C_VEL
LIN {X 0,Y 460.598,Z 125.92,A -85,B 0,C 180,E1 -7935.998,E2 -7935.998} C_VEL
LIN {X 0,Y 460.57,Z 125.926,A -85,B 0,C 180,E1 -7938.902,E2 -7938.902} C_VEL
LIN {X 0,Y 460.514,Z 125.933,A -85,B 0,C 180,E1 -7941.486,E2 -7941.486} C_VEL
LIN {X 0,Y 460.54,Z 125.927,A -85,B 0,C 180,E1 -7944.332,E2 -7944.332} C_VEL
LIN {X 0,Y 460.571,Z 125.926,A -85,B 0,C 180,E1 -7947.244,E2 -7947.244} C_VEL
LIN {X 0,Y 460.509,Z 125.932,A -85,B 0,C 180,E1 -7950.24,E2 -7950.24} C_VEL
LIN {X 0,Y 460.527,Z 125.929,A -85,B 0,C 180,E1 -7953.325,E2 -7953.325} C_VEL
LIN {X 0,Y 460.476,Z 125.942,A -85,B 0,C 180,E1 -7956.529,E2 -7956.529} C_VEL
LIN {X 0,Y 460.523,Z 125.93,A -85,B 0,C 180,E1 -7959.863,E2 -7959.863} C_VEL
LIN {X 0,Y 460.51,Z 125.932,A -85,B 0,C 180,E1 -7962.9,E2 -7962.9} C_VEL
LIN {X 0,Y 460.507,Z 125.933,A -85,B 0,C 180,E1 -7965.831,E2 -7965.831} C_VEL
LIN {X 0,Y 460.529,Z 125.928,A -85,B 0,C 180,E1 -7968.989,E2 -7968.989} C_VEL
LIN {X 0,Y 460.525,Z 125.929,A -85,B 0,C 180,E1 -7971.267,E2 -7971.267} C_VEL
LIN {X 0,Y 460.511,Z 125.931,A -85,B 0,C 180,E1 -7974.555,E2 -7974.555} C_VEL
LIN {X 0,Y 460.529,Z 125.935,A -85,B 0,C 180,E1 -7977.716,E2 -7977.716} C_VEL
LIN {X 0,Y 460.539,Z 125.927,A -85,B 0,C 180,E1 -7980.769,E2 -7980.769} C_VEL
LIN {X 0,Y 460.563,Z 125.93,A -85,B 0,C 180,E1 -7983.735,E2 -7983.735} C_VEL
LIN {X 0,Y 460.597,Z 125.985,A -85,B 0,C 180,E1 -7986.865,E2 -7986.865} C_VEL
LIN {X 0,Y 461.682,Z 133.168,A -85,B 0,C 180,E1 -7988.572,E2 -7988.572} C_VEL
LIN {X 0,Y 461.333,Z 144.562,A -85,B 0,C 180,E1 -7991.072,E2 -7991.072} C_VEL
LIN {X 0,Y 460.721,Z 159.437,A -85,B 0,C 180,E1 -7994.291,E2 -7994.291} C_VEL
LIN {X 0,Y 460.449,Z 169.434,A -85,B 0,C 180,E1 -7996.386,E2 -7996.386} C_VEL
LIN {X 0,Y 461.294,Z 175.605,A -85,B 0,C 180,E1 -7996.545,E2 -7996.545} C_VEL
LIN {X 0,Y 462.585,Z 186.739,A -85,B 0,C 180,E1 -7996.757,E2 -7996.757} C_VEL
LIN {X 0,Y 462.294,Z 245.85,A -85,B 0,C 180,E1 -7997.693,E2 -7997.693} C_VEL
LIN {X 0,Y 462.019,Z 255.481,A -85,B 0,C 180,E1 -7997.955,E2 -7997.955} C_VEL
LIN {X 0,Y 461.743,Z 265.535,A -85,B 0,C 180,E1 -7998.365,E2 -7998.365} C_VEL
LIN {X 0,Y 461.408,Z 276.952,A -85,B 0,C 180,E1 -7999.024,E2 -7999.024} C_VEL
LIN {X 0,Y 461.029,Z 285.54,A -85,B 0,C 180,E1 -7999.682,E2 -7999.682} C_VEL
LIN {X 0,Y 460.643,Z 293.618,A -85,B 0,C 180,E1 -8000.45,E2 -8000.45} C_VEL
LIN {X 0,Y 460.407,Z 300.293,A -85,B 0,C 180,E1 -8001.22,E2 -8001.22} C_VEL
LIN {X 0,Y 460.14,Z 306.628,A -85,B 0,C 180,E1 -8002.099,E2 -8002.099} C_VEL
LIN {X 0,Y 459.943,Z 311.892,A -85,B 0,C 180,E1 -8002.979,E2 -8002.979} C_VEL
LIN {X 0,Y 459.809,Z 316.283,A -85,B 0,C 180,E1 -8003.858,E2 -8003.858} C_VEL
LIN {X 0,Y 459.652,Z 321.457,A -85,B 0,C 180,E1 -8005.176,E2 -8005.176} C_VEL
LIN {X 0,Y 459.622,Z 325.258,A -85,B 0,C 180,E1 -8006.494,E2 -8006.494} C_VEL
LIN {X 0,Y 459.575,Z 327.005,A -85,B 0,C 180,E1 -8007.371,E2 -8007.371} C_VEL
LIN {X 0,Y 459.515,Z 328.256,A -85,B 0,C 180,E1 -8008.247,E2 -8008.247} C_VEL
LIN {X 0,Y 459.492,Z 329.035,A -85,B 0,C 180,E1 -8009.124,E2 -8009.124} C_VEL
LIN {X 0,Y 459.5,Z 329.33,A -85,B 0,C 180,E1 -8010,E2 -8010} C_VEL
LIN {X 0,Y 459.492,Z 329.034,A -85,B 0,C 180,E1 -8010.877,E2 -8010.877} C_VEL
LIN {X 0,Y 459.515,Z 328.252,A -85,B 0,C 180,E1 -8011.753,E2 -8011.753} C_VEL
LIN {X 0,Y 459.575,Z 326.999,A -85,B 0,C 180,E1 -8012.63,E2 -8012.63} C_VEL
LIN {X 0,Y 459.605,Z 324.094,A -85,B 0,C 180,E1 -8013.946,E2 -8013.946} C_VEL
LIN {X 0,Y 459.652,Z 321.447,A -85,B 0,C 180,E1 -8014.824,E2 -8014.824} C_VEL
LIN {X 0,Y 459.802,Z 316.267,A -85,B 0,C 180,E1 -8016.142,E2 -8016.142} C_VEL
LIN {X 0,Y 459.981,Z 309.44,A -85,B 0,C 180,E1 -8017.462,E2 -8017.462} C_VEL
LIN {X 0,Y 460.326,Z 301.978,A -85,B 0,C 180,E1 -8018.561,E2 -8018.561} C_VEL
LIN {X 0,Y 460.586,Z 294.617,A -85,B 0,C 180,E1 -8019.441,E2 -8019.441} C_VEL
LIN {X 0,Y 460.988,Z 286.738,A -85,B 0,C 180,E1 -8020.209,E2 -8020.209} C_VEL
LIN {X 0,Y 461.311,Z 278.41,A -85,B 0,C 180,E1 -8020.867,E2 -8020.867} C_VEL
LIN {X 0,Y 461.696,Z 267.778,A -85,B 0,C 180,E1 -8021.525,E2 -8021.525} C_VEL
LIN {X 0,Y 461.981,Z 256.214,A -85,B 0,C 180,E1 -8022.018,E2 -8022.018} C_VEL
LIN {X 0,Y 462.239,Z 246.543,A -85,B 0,C 180,E1 -8022.29,E2 -8022.29} C_VEL
LIN {X 0,Y 462.527,Z 193.492,A -85,B 0,C 180,E1 -8023.136,E2 -8023.136} C_VEL
LIN {X 0,Y 462.416,Z 183.867,A -85,B 0,C 180,E1 -8023.29,E2 -8023.29} C_VEL
LIN {X 0,Y 460.45,Z 169.67,A -85,B 0,C 180,E1 -8023.592,E2 -8023.592} C_VEL
LIN {X 0,Y 460.524,Z 166.757,A -85,B 0,C 180,E1 -8024.133,E2 -8024.133} C_VEL
LIN {X 0,Y 461.039,Z 151.022,A -85,B 0,C 180,E1 -8027.522,E2 -8027.522} C_VEL
LIN {X 0,Y 461.634,Z 137.358,A -85,B 0,C 180,E1 -8030.497,E2 -8030.497} C_VEL
LIN {X 0,Y 461.569,Z 131.722,A -85,B 0,C 180,E1 -8031.751,E2 -8031.751} C_VEL
LIN {X 0,Y 460.598,Z 125.974,A -85,B 0,C 180,E1 -8033.136,E2 -8033.136} C_VEL
LIN {X 0,Y 460.564,Z 125.93,A -85,B 0,C 180,E1 -8036.265,E2 -8036.265} C_VEL
LIN {X 0,Y 460.54,Z 125.926,A -85,B 0,C 180,E1 -8039.231,E2 -8039.231} C_VEL
LIN {X 0,Y 460.532,Z 125.935,A -85,B 0,C 180,E1 -8042.284,E2 -8042.284} C_VEL
LIN {X 0,Y 460.511,Z 125.931,A -85,B 0,C 180,E1 -8045.446,E2 -8045.446} C_VEL
LIN {X 0,Y 460.545,Z 125.926,A -85,B 0,C 180,E1 -8048.898,E2 -8048.898} C_VEL
LIN {X 0,Y 460.523,Z 125.932,A -85,B 0,C 180,E1 -8052.181,E2 -8052.181} C_VEL
LIN {X 0,Y 460.513,Z 125.933,A -85,B 0,C 180,E1 -8055.411,E2 -8055.411} C_VEL
LIN {X 0,Y 460.532,Z 125.928,A -85,B 0,C 180,E1 -8058.398,E2 -8058.398} C_VEL
LIN {X 0,Y 460.519,Z 125.933,A -85,B 0,C 180,E1 -8061.266,E2 -8061.266} C_VEL
LIN {X 0,Y 460.514,Z 125.93,A -85,B 0,C 180,E1 -8064.555,E2 -8064.555} C_VEL
LIN {X 0,Y 460.532,Z 125.93,A -85,B 0,C 180,E1 -8067.716,E2 -8067.716} C_VEL
LIN {X 0,Y 460.541,Z 125.929,A -85,B 0,C 180,E1 -8070.769,E2 -8070.769} C_VEL
LIN {X 0,Y 460.564,Z 125.924,A -85,B 0,C 180,E1 -8073.735,E2 -8073.735} C_VEL
LIN {X 0,Y 460.547,Z 125.929,A -85,B 0,C 180,E1 -8076.624,E2 -8076.624} C_VEL
LIN {X 0,Y 460.552,Z 125.926,A -85,B 0,C 180,E1 -8079.453,E2 -8079.453} C_VEL
LIN {X 0,Y 460.561,Z 125.926,A -85,B 0,C 180,E1 -8082.23,E2 -8082.23} C_VEL
LIN {X 0,Y 460.567,Z 125.927,A -85,B 0,C 180,E1 -8084.965,E2 -8084.965} C_VEL
LIN {X 0,Y 460.612,Z 125.925,A -85,B 0,C 180,E1 -8088.559,E2 -8088.559} C_VEL
LIN {X 0,Y 460.697,Z 125.911,A -85,B 0,C 180,E1 -8092.109,E2 -8092.109} C_VEL
LIN {X 0,Y 460.696,Z 125.909,A -85,B 0,C 180,E1 -8094.748,E2 -8094.748} C_VEL
LIN {X 0,Y 460.801,Z 125.894,A -85,B 0,C 180,E1 -8097.378,E2 -8097.378} C_VEL
LIN {X 0,Y 460.854,Z 125.894,A -85,B 0,C 180,E1 -8100,E2 -8100} C_VEL
LIN {X 0,Y 460.801,Z 125.895,A -85,B 0,C 180,E1 -8102.623,E2 -8102.623} C_VEL
LIN {X 0,Y 460.711,Z 125.909,A -85,B 0,C 180,E1 -8106.13,E2 -8106.13} C_VEL
LIN {X 0,Y 460.63,Z 125.915,A -85,B 0,C 180,E1 -8108.776,E2 -8108.776} C_VEL
LIN {X 0,Y 460.636,Z 125.915,A -85,B 0,C 180,E1 -8112.457,E2 -8112.457} C_VEL
LIN {X 0,Y 460.602,Z 125.92,A -85,B 0,C 180,E1 -8115.998,E2 -8115.998} C_VEL
LIN {X 0,Y 460.572,Z 125.925,A -85,B 0,C 180,E1 -8118.902,E2 -8118.902} C_VEL
LIN {X 0,Y 460.517,Z 125.934,A -85,B 0,C 180,E1 -8121.486,E2 -8121.486} C_VEL
LIN {X 0,Y 460.542,Z 125.926,A -85,B 0,C 180,E1 -8124.332,E2 -8124.332} C_VEL
LIN {X 0,Y 460.575,Z 125.927,A -85,B 0,C 180,E1 -8127.244,E2 -8127.244} C_VEL
LIN {X 0,Y 460.512,Z 125.931,A -85,B 0,C 180,E1 -8130.24,E2 -8130.24} C_VEL
LIN {X 0,Y 460.531,Z 125.929,A -85,B 0,C 180,E1 -8133.325,E2 -8133.325} C_VEL
LIN {X 0,Y 460.48,Z 125.939,A -85,B 0,C 180,E1 -8136.529,E2 -8136.529} C_VEL
LIN {X 0,Y 460.527,Z 125.929,A -85,B 0,C 180,E1 -8139.863,E2 -8139.863} C_VEL
LIN {X 0,Y 460.513,Z 125.932,A -85,B 0,C 180,E1 -8142.9,E2 -8142.9} C_VEL
LIN {X 0,Y 460.51,Z 125.932,A -85,B 0,C 180,E1 -8145.831,E2 -8145.831} C_VEL
LIN {X 0,Y 460.533,Z 125.928,A -85,B 0,C 180,E1 -8148.989,E2 -8148.989} C_VEL
LIN {X 0,Y 460.528,Z 125.928,A -85,B 0,C 180,E1 -8151.267,E2 -8151.267} C_VEL
LIN {X 0,Y 460.514,Z 125.931,A -85,B 0,C 180,E1 -8154.555,E2 -8154.555} C_VEL
LIN {X 0,Y 460.532,Z 125.933,A -85,B 0,C 180,E1 -8157.716,E2 -8157.716} C_VEL
LIN {X 0,Y 460.542,Z 125.926,A -85,B 0,C 180,E1 -8160.769,E2 -8160.769} C_VEL
LIN {X 0,Y 460.558,Z 125.931,A -85,B 0,C 180,E1 -8163.734,E2 -8163.734} C_VEL
LIN {X 0,Y 460.547,Z 125.928,A -85,B 0,C 180,E1 -8166.624,E2 -8166.624} C_VEL
LIN {X 0,Y 460.662,Z 126.076,A -85,B 0,C 180,E1 -8169.807,E2 -8169.807} C_VEL
LIN {X 0,Y 461.184,Z 132.092,A -85,B 0,C 180,E1 -8171.336,E2 -8171.336} C_VEL
LIN {X 0,Y 460.76,Z 145.307,A -85,B 0,C 180,E1 -8174.518,E2 -8174.518} C_VEL
LIN {X 0,Y 460.595,Z 150.702,A -85,B 0,C 180,E1 -8175.792,E2 -8175.792} C_VEL
LIN {X 0,Y 460.273,Z 152.413,A -85,B 0,C 180,E1 -8176.057,E2 -8176.057} C_VEL
LIN {X 0,Y 459.229,Z 155.461,A -85,B 0,C 180,E1 -8176.293,E2 -8176.293} C_VEL
LIN {X 0,Y 457.56,Z 159.94,A -85,B 0,C 180,E1 -8176.451,E2 -8176.451} C_VEL
LIN {X 0,Y 456.465,Z 163.759,A -85,B 0,C 180,E1 -8176.517,E2 -8176.517} C_VEL
LIN {X 0,Y 455.287,Z 170.164,A -85,B 0,C 180,E1 -8176.583,E2 -8176.583} C_VEL
LIN {X 0,Y 455.429,Z 176.65,A -85,B 0,C 180,E1 -8176.689,E2 -8176.689} C_VEL
LIN {X 0,Y 455.694,Z 180.975,A -85,B 0,C 180,E1 -8176.767,E2 -8176.767} C_VEL
LIN {X 0,Y 455.403,Z 229.546,A -85,B 0,C 180,E1 -8177.551,E2 -8177.551} C_VEL
LIN {X 0,Y 455.245,Z 238.656,A -85,B 0,C 180,E1 -8177.801,E2 -8177.801} C_VEL
LIN {X 0,Y 455.017,Z 248.255,A -85,B 0,C 180,E1 -8178.191,E2 -8178.191} C_VEL
LIN {X 0,Y 454.724,Z 256.431,A -85,B 0,C 180,E1 -8178.635,E2 -8178.635} C_VEL
LIN {X 0,Y 454.382,Z 266.035,A -85,B 0,C 180,E1 -8179.303,E2 -8179.303} C_VEL
LIN {X 0,Y 453.998,Z 275.851,A -85,B 0,C 180,E1 -8180.196,E2 -8180.196} C_VEL
LIN {X 0,Y 453.593,Z 283.591,A -85,B 0,C 180,E1 -8181.086,E2 -8181.086} C_VEL
LIN {X 0,Y 453.277,Z 289.954,A -85,B 0,C 180,E1 -8181.978,E2 -8181.978} C_VEL
LIN {X 0,Y 453.098,Z 295.241,A -85,B 0,C 180,E1 -8182.872,E2 -8182.872} C_VEL
LIN {X 0,Y 452.978,Z 299.655,A -85,B 0,C 180,E1 -8183.765,E2 -8183.765} C_VEL
LIN {X 0,Y 452.667,Z 304.847,A -85,B 0,C 180,E1 -8185.101,E2 -8185.101} C_VEL
LIN {X 0,Y 452.673,Z 307.512,A -85,B 0,C 180,E1 -8185.994,E2 -8185.994} C_VEL
LIN {X 0,Y 452.529,Z 310.433,A -85,B 0,C 180,E1 -8187.329,E2 -8187.329} C_VEL
LIN {X 0,Y 452.438,Z 311.712,A -85,B 0,C 180,E1 -8188.219,E2 -8188.219} C_VEL
LIN {X 0,Y 452.403,Z 312.521,A -85,B 0,C 180,E1 -8189.11,E2 -8189.11} C_VEL
LIN {X 0,Y 452.407,Z 312.829,A -85,B 0,C 180,E1 -8190,E2 -8190} C_VEL
LIN {X 0,Y 452.403,Z 312.555,A -85,B 0,C 180,E1 -8190.89,E2 -8190.89} C_VEL
LIN {X 0,Y 452.438,Z 311.814,A -85,B 0,C 180,E1 -8191.78,E2 -8191.78} C_VEL
LIN {X 0,Y 452.528,Z 310.603,A -85,B 0,C 180,E1 -8192.67,E2 -8192.67} C_VEL
LIN {X 0,Y 452.662,Z 307.754,A -85,B 0,C 180,E1 -8194.006,E2 -8194.006} C_VEL
LIN {X 0,Y 452.661,Z 305.165,A -85,B 0,C 180,E1 -8194.898,E2 -8194.898} C_VEL
LIN {X 0,Y 452.965,Z 300.058,A -85,B 0,C 180,E1 -8196.235,E2 -8196.235} C_VEL
LIN {X 0,Y 453.099,Z 294.568,A -85,B 0,C 180,E1 -8197.352,E2 -8197.352} C_VEL
LIN {X 0,Y 453.418,Z 287.673,A -85,B 0,C 180,E1 -8198.467,E2 -8198.467} C_VEL
LIN {X 0,Y 453.78,Z 279.753,A -85,B 0,C 180,E1 -8199.471,E2 -8199.471} C_VEL
LIN {X 0,Y 454.108,Z 272.201,A -85,B 0,C 180,E1 -8200.252,E2 -8200.252} C_VEL
LIN {X 0,Y 454.432,Z 264.287,A -85,B 0,C 180,E1 -8200.921,E2 -8200.921} C_VEL
LIN {X 0,Y 454.792,Z 256.117,A -85,B 0,C 180,E1 -8201.476,E2 -8201.476} C_VEL
LIN {X 0,Y 455.028,Z 247.848,A -85,B 0,C 180,E1 -8201.922,E2 -8201.922} C_VEL
LIN {X 0,Y 455.293,Z 238.927,A -85,B 0,C 180,E1 -8202.282,E2 -8202.282} C_VEL
LIN {X 0,Y 455.471,Z 229.942,A -85,B 0,C 180,E1 -8202.532,E2 -8202.532} C_VEL
LIN {X 0,Y 455.731,Z 167.402,A -85,B 0,C 180,E1 -8203.542,E2 -8203.542} C_VEL
LIN {X 0,Y 453.577,Z 154.136,A -85,B 0,C 180,E1 -8203.842,E2 -8203.842} C_VEL
LIN {X 0,Y 453.515,Z 152.979,A -85,B 0,C 180,E1 -8204.015,E2 -8204.015} C_VEL
LIN {X 0,Y 453.949,Z 140.106,A -85,B 0,C 180,E1 -8207.107,E2 -8207.107} C_VEL
LIN {X 0,Y 454.147,Z 131.33,A -85,B 0,C 180,E1 -8209.268,E2 -8209.268} C_VEL
LIN {X 0,Y 453.577,Z 126.893,A -85,B 0,C 180,E1 -8210.462,E2 -8210.462} C_VEL
LIN {X 0,Y 453.494,Z 126.806,A -85,B 0,C 180,E1 -8213.886,E2 -8213.886} C_VEL
LIN {X 0,Y 453.503,Z 126.807,A -85,B 0,C 180,E1 -8216.706,E2 -8216.706} C_VEL
LIN {X 0,Y 453.475,Z 126.808,A -85,B 0,C 180,E1 -8219.731,E2 -8219.731} C_VEL
LIN {X 0,Y 453.489,Z 126.805,A -85,B 0,C 180,E1 -8223.189,E2 -8223.189} C_VEL
LIN {X 0,Y 453.455,Z 126.813,A -85,B 0,C 180,E1 -8226.299,E2 -8226.299} C_VEL
LIN {X 0,Y 453.516,Z 126.804,A -85,B 0,C 180,E1 -8229.447,E2 -8229.447} C_VEL
LIN {X 0,Y 453.462,Z 126.809,A -85,B 0,C 180,E1 -8232.995,E2 -8232.995} C_VEL
LIN {X 0,Y 453.463,Z 126.814,A -85,B 0,C 180,E1 -8235.778,E2 -8235.778} C_VEL
LIN {X 0,Y 453.478,Z 126.807,A -85,B 0,C 180,E1 -8238.209,E2 -8238.209} C_VEL
LIN {X 0,Y 453.486,Z 126.806,A -85,B 0,C 180,E1 -8240.794,E2 -8240.794} C_VEL
LIN {X 0,Y 453.456,Z 126.81,A -85,B 0,C 180,E1 -8243.917,E2 -8243.917} C_VEL
LIN {X 0,Y 453.482,Z 126.812,A -85,B 0,C 180,E1 -8247.151,E2 -8247.151} C_VEL
LIN {X 0,Y 453.474,Z 126.807,A -85,B 0,C 180,E1 -8250.268,E2 -8250.268} C_VEL
LIN {X 0,Y 453.506,Z 126.807,A -85,B 0,C 180,E1 -8253.294,E2 -8253.294} C_VEL
LIN {X 0,Y 453.501,Z 126.804,A -85,B 0,C 180,E1 -8256.239,E2 -8256.239} C_VEL
LIN {X 0,Y 453.482,Z 126.809,A -85,B 0,C 180,E1 -8259.117,E2 -8259.117} C_VEL
LIN {X 0,Y 453.51,Z 126.803,A -85,B 0,C 180,E1 -8261.944,E2 -8261.944} C_VEL
LIN {X 0,Y 453.538,Z 126.804,A -85,B 0,C 180,E1 -8264.726,E2 -8264.726} C_VEL
LIN {X 0,Y 453.601,Z 126.791,A -85,B 0,C 180,E1 -8267.472,E2 -8267.472} C_VEL
LIN {X 0,Y 453.591,Z 126.792,A -85,B 0,C 180,E1 -8271.087,E2 -8271.087} C_VEL
LIN {X 0,Y 453.676,Z 126.784,A -85,B 0,C 180,E1 -8273.775,E2 -8273.775} C_VEL
LIN {X 0,Y 453.763,Z 126.771,A -85,B 0,C 180,E1 -8277.337,E2 -8277.337} C_VEL
LIN {X 0,Y 453.823,Z 126.771,A -85,B 0,C 180,E1 -8280,E2 -8280} C_VEL
LIN {X 0,Y 453.743,Z 126.773,A -85,B 0,C 180,E1 -8282.663,E2 -8282.663} C_VEL
LIN {X 0,Y 453.676,Z 126.784,A -85,B 0,C 180,E1 -8286.225,E2 -8286.225} C_VEL
LIN {X 0,Y 453.59,Z 126.793,A -85,B 0,C 180,E1 -8288.913,E2 -8288.913} C_VEL
LIN {X 0,Y 453.562,Z 126.796,A -85,B 0,C 180,E1 -8292.529,E2 -8292.529} C_VEL
LIN {X 0,Y 453.543,Z 126.798,A -85,B 0,C 180,E1 -8296.196,E2 -8296.196} C_VEL
LIN {X 0,Y 453.519,Z 126.806,A -85,B 0,C 180,E1 -8299.041,E2 -8299.041} C_VEL
LIN {X 0,Y 453.474,Z 126.807,A -85,B 0,C 180,E1 -8301.836,E2 -8301.836} C_VEL
LIN {X 0,Y 453.511,Z 126.806,A -85,B 0,C 180,E1 -8304.734,E2 -8304.734} C_VEL
LIN {X 0,Y 453.53,Z 126.8,A -85,B 0,C 180,E1 -8307.96,E2 -8307.96} C_VEL
LIN {X 0,Y 453.464,Z 126.808,A -85,B 0,C 180,E1 -8311.525,E2 -8311.525} C_VEL
LIN {X 0,Y 453.487,Z 126.811,A -85,B 0,C 180,E1 -8314.778,E2 -8314.778} C_VEL
LIN {X 0,Y 453.459,Z 126.814,A -85,B 0,C 180,E1 -8318.312,E2 -8318.312} C_VEL
LIN {X 0,Y 453.492,Z 126.81,A -85,B 0,C 180,E1 -8320.609,E2 -8320.609} C_VEL
LIN {X 0,Y 453.452,Z 126.809,A -85,B 0,C 180,E1 -8323.244,E2 -8323.244} C_VEL
LIN {X 0,Y 453.462,Z 126.811,A -85,B 0,C 180,E1 -8325.779,E2 -8325.779} C_VEL
LIN {X 0,Y 453.478,Z 126.813,A -85,B 0,C 180,E1 -8328.21,E2 -8328.21} C_VEL
LIN {X 0,Y 453.493,Z 126.805,A -85,B 0,C 180,E1 -8330.794,E2 -8330.794} C_VEL
LIN {X 0,Y 453.455,Z 126.817,A -85,B 0,C 180,E1 -8333.918,E2 -8333.918} C_VEL
LIN {X 0,Y 453.48,Z 126.807,A -85,B 0,C 180,E1 -8337.151,E2 -8337.151} C_VEL
LIN {X 0,Y 453.474,Z 126.808,A -85,B 0,C 180,E1 -8340.269,E2 -8340.269} C_VEL
LIN {X 0,Y 453.506,Z 126.807,A -85,B 0,C 180,E1 -8343.294,E2 -8343.294} C_VEL
LIN {X 0,Y 453.543,Z 126.887,A -85,B 0,C 180,E1 -8346.725,E2 -8346.725} C_VEL
LIN {X 0,Y 454.697,Z 134.096,A -85,B 0,C 180,E1 -8348.464,E2 -8348.464} C_VEL
LIN {X 0,Y 454.396,Z 143.856,A -85,B 0,C 180,E1 -8350.642,E2 -8350.642} C_VEL
LIN {X 0,Y 453.74,Z 158.823,A -85,B 0,C 180,E1 -8353.935,E2 -8353.935} C_VEL
LIN {X 0,Y 453.408,Z 169.308,A -85,B 0,C 180,E1 -8356.17,E2 -8356.17} C_VEL
LIN {X 0,Y 454.216,Z 175.146,A -85,B 0,C 180,E1 -8356.326,E2 -8356.326} C_VEL
LIN {X 0,Y 455.688,Z 187.603,A -85,B 0,C 180,E1 -8356.568,E2 -8356.568} C_VEL
LIN {X 0,Y 455.379,Z 245.777,A -85,B 0,C 180,E1 -8357.504,E2 -8357.504} C_VEL
LIN {X 0,Y 455.086,Z 255.361,A -85,B 0,C 180,E1 -8357.769,E2 -8357.769} C_VEL
LIN {X 0,Y 454.795,Z 265.412,A -85,B 0,C 180,E1 -8358.185,E2 -8358.185} C_VEL
LIN {X 0,Y 454.441,Z 276.828,A -85,B 0,C 180,E1 -8358.854,E2 -8358.854} C_VEL
LIN {X 0,Y 454.052,Z 285.415,A -85,B 0,C 180,E1 -8359.521,E2 -8359.521} C_VEL
LIN {X 0,Y 453.634,Z 293.492,A -85,B 0,C 180,E1 -8360.301,E2 -8360.301} C_VEL
LIN {X 0,Y 453.391,Z 300.167,A -85,B 0,C 180,E1 -8361.083,E2 -8361.083} C_VEL
LIN {X 0,Y 453.093,Z 306.501,A -85,B 0,C 180,E1 -8361.976,E2 -8361.976} C_VEL
LIN {X 0,Y 452.887,Z 311.765,A -85,B 0,C 180,E1 -8362.869,E2 -8362.869} C_VEL
LIN {X 0,Y 452.721,Z 316.155,A -85,B 0,C 180,E1 -8363.762,E2 -8363.762} C_VEL
LIN {X 0,Y 452.583,Z 321.33,A -85,B 0,C 180,E1 -8365.101,E2 -8365.101} C_VEL
LIN {X 0,Y 452.519,Z 325.13,A -85,B 0,C 180,E1 -8366.439,E2 -8366.439} C_VEL
LIN {X 0,Y 452.501,Z 326.877,A -85,B 0,C 180,E1 -8367.33,E2 -8367.33} C_VEL
LIN {X 0,Y 452.432,Z 328.128,A -85,B 0,C 180,E1 -8368.22,E2 -8368.22} C_VEL
LIN {X 0,Y 452.401,Z 328.907,A -85,B 0,C 180,E1 -8369.11,E2 -8369.11} C_VEL
LIN {X 0,Y 452.405,Z 329.202,A -85,B 0,C 180,E1 -8370,E2 -8370} C_VEL
LIN {X 0,Y 452.401,Z 328.905,A -85,B 0,C 180,E1 -8370.89,E2 -8370.89} C_VEL
LIN {X 0,Y 452.432,Z 328.124,A -85,B 0,C 180,E1 -8371.781,E2 -8371.781} C_VEL
LIN {X 0,Y 452.501,Z 326.87,A -85,B 0,C 180,E1 -8372.671,E2 -8372.671} C_VEL
LIN {X 0,Y 452.505,Z 323.965,A -85,B 0,C 180,E1 -8374.008,E2 -8374.008} C_VEL
LIN {X 0,Y 452.583,Z 321.318,A -85,B 0,C 180,E1 -8374.9,E2 -8374.9} C_VEL
LIN {X 0,Y 452.729,Z 316.137,A -85,B 0,C 180,E1 -8376.239,E2 -8376.239} C_VEL
LIN {X 0,Y 452.915,Z 309.309,A -85,B 0,C 180,E1 -8377.579,E2 -8377.579} C_VEL
LIN {X 0,Y 453.285,Z 301.847,A -85,B 0,C 180,E1 -8378.695,E2 -8378.695} C_VEL
LIN {X 0,Y 453.575,Z 294.486,A -85,B 0,C 180,E1 -8379.589,E2 -8379.589} C_VEL
LIN {X 0,Y 453.992,Z 286.606,A -85,B 0,C 180,E1 -8380.368,E2 -8380.368} C_VEL
LIN {X 0,Y 454.326,Z 278.278,A -85,B 0,C 180,E1 -8381.036,E2 -8381.036} C_VEL
LIN {X 0,Y 454.74,Z 267.644,A -85,B 0,C 180,E1 -8381.704,E2 -8381.704} C_VEL
LIN {X 0,Y 455.057,Z 256.077,A -85,B 0,C 180,E1 -8382.204,E2 -8382.204} C_VEL
LIN {X 0,Y 455.302,Z 246.401,A -85,B 0,C 180,E1 -8382.48,E2 -8382.48} C_VEL
LIN {X 0,Y 455.599,Z 199.568,A -85,B 0,C 180,E1 -8383.241,E2 -8383.241} C_VEL
LIN {X 0,Y 455.516,Z 184.432,A -85,B 0,C 180,E1 -8383.484,E2 -8383.484} C_VEL
LIN {X 0,Y 453.438,Z 169.535,A -85,B 0,C 180,E1 -8383.806,E2 -8383.806} C_VEL
LIN {X 0,Y 453.5,Z 166.627,A -85,B 0,C 180,E1 -8384.357,E2 -8384.357} C_VEL
LIN {X 0,Y 454.059,Z 150.895,A -85,B 0,C 180,E1 -8387.8,E2 -8387.8} C_VEL
LIN {X 0,Y 454.67,Z 137.232,A -85,B 0,C 180,E1 -8390.825,E2 -8390.825} C_VEL
LIN {X 0,Y 454.509,Z 132.455,A -85,B 0,C 180,E1 -8391.91,E2 -8391.91} C_VEL
LIN {X 0,Y 453.544,Z 126.873,A -85,B 0,C 180,E1 -8393.275,E2 -8393.275} C_VEL
LIN {X 0,Y 453.507,Z 126.807,A -85,B 0,C 180,E1 -8396.706,E2 -8396.706} C_VEL
LIN {X 0,Y 453.473,Z 126.808,A -85,B 0,C 180,E1 -8399.785,E2 -8399.785} C_VEL
LIN {X 0,Y 453.491,Z 126.804,A -85,B 0,C 180,E1 -8403.189,E2 -8403.189} C_VEL
LIN {X 0,Y 453.454,Z 126.814,A -85,B 0,C 180,E1 -8406.299,E2 -8406.299} C_VEL
LIN {X 0,Y 453.49,Z 126.806,A -85,B 0,C 180,E1 -8409.45,E2 -8409.45} C_VEL
LIN {X 0,Y 453.477,Z 126.813,A -85,B 0,C 180,E1 -8411.935,E2 -8411.935} C_VEL
LIN {X 0,Y 453.484,Z 126.81,A -85,B 0,C 180,E1 -8415.471,E2 -8415.471} C_VEL
LIN {X 0,Y 453.48,Z 126.807,A -85,B 0,C 180,E1 -8418.209,E2 -8418.209} C_VEL
LIN {X 0,Y 453.488,Z 126.805,A -85,B 0,C 180,E1 -8420.795,E2 -8420.795} C_VEL
LIN {X 0,Y 453.457,Z 126.811,A -85,B 0,C 180,E1 -8423.918,E2 -8423.918} C_VEL
LIN {X 0,Y 453.484,Z 126.811,A -85,B 0,C 180,E1 -8427.151,E2 -8427.151} C_VEL
LIN {X 0,Y 453.476,Z 126.806,A -85,B 0,C 180,E1 -8430.268,E2 -8430.268} C_VEL
LIN {X 0,Y 453.508,Z 126.807,A -85,B 0,C 180,E1 -8433.294,E2 -8433.294} C_VEL
LIN {X 0,Y 453.504,Z 126.803,A -85,B 0,C 180,E1 -8436.239,E2 -8436.239} C_VEL
LIN {X 0,Y 453.484,Z 126.81,A -85,B 0,C 180,E1 -8439.118,E2 -8439.118} C_VEL
LIN {X 0,Y 453.513,Z 126.802,A -85,B 0,C 180,E1 -8441.945,E2 -8441.945} C_VEL
LIN {X 0,Y 453.541,Z 126.805,A -85,B 0,C 180,E1 -8444.726,E2 -8444.726} C_VEL
LIN {X 0,Y 453.561,Z 126.802,A -85,B 0,C 180,E1 -8448.379,E2 -8448.379} C_VEL
LIN {X 0,Y 453.654,Z 126.787,A -85,B 0,C 180,E1 -8451.985,E2 -8451.985} C_VEL
LIN {X 0,Y 453.669,Z 126.785,A -85,B 0,C 180,E1 -8454.667,E2 -8454.667} C_VEL
LIN {X 0,Y 453.745,Z 126.773,A -85,B 0,C 180,E1 -8457.337,E2 -8457.337} C_VEL
LIN {X 0,Y 453.824,Z 126.77,A -85,B 0,C 180,E1 -8460,E2 -8460} C_VEL
LIN {X 0,Y 453.745,Z 126.774,A -85,B 0,C 180,E1 -8462.663,E2 -8462.663} C_VEL
LIN {X 0,Y 453.679,Z 126.784,A -85,B 0,C 180,E1 -8466.225,E2 -8466.225} C_VEL
LIN {X 0,Y 453.594,Z 126.792,A -85,B 0,C 180,E1 -8468.913,E2 -8468.913} C_VEL
LIN {X 0,Y 453.604,Z 126.79,A -85,B 0,C 180,E1 -8472.551,E2 -8472.551} C_VEL
LIN {X 0,Y 453.547,Z 126.798,A -85,B 0,C 180,E1 -8476.196,E2 -8476.196} C_VEL
LIN {X 0,Y 453.522,Z 126.804,A -85,B 0,C 180,E1 -8479.041,E2 -8479.041} C_VEL
LIN {X 0,Y 453.478,Z 126.807,A -85,B 0,C 180,E1 -8481.836,E2 -8481.836} C_VEL
LIN {X 0,Y 453.514,Z 126.804,A -85,B 0,C 180,E1 -8484.735,E2 -8484.735} C_VEL
LIN {X 0,Y 453.534,Z 126.799,A -85,B 0,C 180,E1 -8487.96,E2 -8487.96} C_VEL
LIN {X 0,Y 453.467,Z 126.808,A -85,B 0,C 180,E1 -8491.525,E2 -8491.525} C_VEL
LIN {X 0,Y 453.491,Z 126.812,A -85,B 0,C 180,E1 -8494.778,E2 -8494.778} C_VEL
LIN {X 0,Y 453.462,Z 126.812,A -85,B 0,C 180,E1 -8498.312,E2 -8498.312} C_VEL
LIN {X 0,Y 453.495,Z 126.811,A -85,B 0,C 180,E1 -8500.609,E2 -8500.609} C_VEL
LIN {X 0,Y 453.454,Z 126.809,A -85,B 0,C 180,E1 -8503.244,E2 -8503.244} C_VEL
LIN {X 0,Y 453.465,Z 126.809,A -85,B 0,C 180,E1 -8505.779,E2 -8505.779} C_VEL
LIN {X 0,Y 453.481,Z 126.813,A -85,B 0,C 180,E1 -8508.209,E2 -8508.209} C_VEL
LIN {X 0,Y 453.517,Z 126.802,A -85,B 0,C 180,E1 -8510.79,E2 -8510.79} C_VEL
LIN {X 0,Y 453.458,Z 126.815,A -85,B 0,C 180,E1 -8513.917,E2 -8513.917} C_VEL
LIN {X 0,Y 453.483,Z 126.806,A -85,B 0,C 180,E1 -8517.151,E2 -8517.151} C_VEL
LIN {X 0,Y 453.477,Z 126.809,A -85,B 0,C 180,E1 -8520.268,E2 -8520.268} C_VEL
LIN {X 0,Y 453.504,Z 126.806,A -85,B 0,C 180,E1 -8523.294,E2 -8523.294} C_VEL
LIN {X 0,Y 453.5,Z 126.807,A -85,B 0,C 180,E1 -8526.238,E2 -8526.238} C_VEL
LIN {X 0,Y 453.604,Z 127.036,A -85,B 0,C 180,E1 -8529.716,E2 -8529.716} C_VEL
LIN {X 0,Y 454.191,Z 132.162,A -85,B 0,C 180,E1 -8531.037,E2 -8531.037} C_VEL
LIN {X 0,Y 453.814,Z 143.509,A -85,B 0,C 180,E1 -8533.814,E2 -8533.814} C_VEL
LIN {X 0,Y 453.521,Z 153.551,A -85,B 0,C 180,E1 -8536.196,E2 -8536.196} C_VEL
LIN {X 0,Y 453.729,Z 155.251,A -85,B 0,C 180,E1 -8536.297,E2 -8536.297} C_VEL
LIN {X 0,Y 455.789,Z 168.757,A -85,B 0,C 180,E1 -8536.576,E2 -8536.576} C_VEL
LIN {X 0,Y 455.694,Z 180.975,A -85,B 0,C 180,E1 -8536.767,E2 -8536.767} C_VEL
LIN {X 0,Y 454.995,Z 186.813,A -85,B 0,C 180,E1 -8536.838,E2 -8536.838} C_VEL
LIN {X 0,Y 449.419,Z 205.807,A -85,B 0,C 180,E1 -8536.976,E2 -8536.976} C_VEL
LIN {X 0,Y 448.637,Z 211.646,A -85,B 0,C 180,E1 -8537.046,E2 -8537.046} C_VEL
LIN {X 0,Y 448.477,Z 232.287,A -85,B 0,C 180,E1 -8537.413,E2 -8537.413} C_VEL
LIN {X 0,Y 448.174,Z 244.767,A -85,B 0,C 180,E1 -8537.835,E2 -8537.835} C_VEL
LIN {X 0,Y 447.811,Z 254.697,A -85,B 0,C 180,E1 -8538.342,E2 -8538.342} C_VEL
LIN {X 0,Y 447.586,Z 263.171,A -85,B 0,C 180,E1 -8538.91,E2 -8538.91} C_VEL
LIN {X 0,Y 447.225,Z 270.085,A -85,B 0,C 180,E1 -8539.474,E2 -8539.474} C_VEL
LIN {X 0,Y 446.913,Z 278.021,A -85,B 0,C 180,E1 -8540.267,E2 -8540.267} C_VEL
LIN {X 0,Y 446.591,Z 283.723,A -85,B 0,C 180,E1 -8540.946,E2 -8540.946} C_VEL
LIN {X 0,Y 446.234,Z 290.085,A -85,B 0,C 180,E1 -8541.851,E2 -8541.851} C_VEL
LIN {X 0,Y 446.062,Z 295.372,A -85,B 0,C 180,E1 -8542.759,E2 -8542.759} C_VEL
LIN {X 0,Y 445.927,Z 299.785,A -85,B 0,C 180,E1 -8543.666,E2 -8543.666} C_VEL
LIN {X 0,Y 445.6,Z 304.977,A -85,B 0,C 180,E1 -8545.023,E2 -8545.023} C_VEL
LIN {X 0,Y 445.573,Z 307.642,A -85,B 0,C 180,E1 -8545.93,E2 -8545.93} C_VEL
LIN {X 0,Y 445.459,Z 310.561,A -85,B 0,C 180,E1 -8547.287,E2 -8547.287} C_VEL
LIN {X 0,Y 445.358,Z 311.841,A -85,B 0,C 180,E1 -8548.191,E2 -8548.191} C_VEL
LIN {X 0,Y 445.315,Z 312.65,A -85,B 0,C 180,E1 -8549.095,E2 -8549.095} C_VEL
LIN {X 0,Y 445.316,Z 312.958,A -85,B 0,C 180,E1 -8550,E2 -8550} C_VEL
LIN {X 0,Y 445.315,Z 312.683,A -85,B 0,C 180,E1 -8550.904,E2 -8550.904} C_VEL
LIN {X 0,Y 445.358,Z 311.941,A -85,B 0,C 180,E1 -8551.808,E2 -8551.808} C_VEL
LIN {X 0,Y 445.458,Z 310.73,A -85,B 0,C 180,E1 -8552.713,E2 -8552.713} C_VEL
LIN {X 0,Y 445.561,Z 307.882,A -85,B 0,C 180,E1 -8554.07,E2 -8554.07} C_VEL
LIN {X 0,Y 445.594,Z 305.292,A -85,B 0,C 180,E1 -8554.976,E2 -8554.976} C_VEL
LIN {X 0,Y 445.916,Z 300.185,A -85,B 0,C 180,E1 -8556.334,E2 -8556.334} C_VEL
LIN {X 0,Y 446.11,Z 293.482,A -85,B 0,C 180,E1 -8557.695,E2 -8557.695} C_VEL
LIN {X 0,Y 446.457,Z 286.123,A -85,B 0,C 180,E1 -8558.829,E2 -8558.829} C_VEL
LIN {X 0,Y 446.844,Z 278.859,A -85,B 0,C 180,E1 -8559.734,E2 -8559.734} C_VEL
LIN {X 0,Y 447.173,Z 271.098,A -85,B 0,C 180,E1 -8560.527,E2 -8560.527} C_VEL
LIN {X 0,Y 447.53,Z 262.911,A -85,B 0,C 180,E1 -8561.206,E2 -8561.206} C_VEL
LIN {X 0,Y 447.851,Z 254.368,A -85,B 0,C 180,E1 -8561.771,E2 -8561.771} C_VEL
LIN {X 0,Y 448.295,Z 243.073,A -85,B 0,C 180,E1 -8562.333,E2 -8562.333} C_VEL
LIN {X 0,Y 448.545,Z 231.831,A -85,B 0,C 180,E1 -8562.69,E2 -8562.69} C_VEL
LIN {X 0,Y 448.6,Z 209.793,A -85,B 0,C 180,E1 -8563.079,E2 -8563.079} C_VEL
LIN {X 0,Y 448.802,Z 167.901,A -85,B 0,C 180,E1 -8563.749,E2 -8563.749} C_VEL
LIN {X 0,Y 446.568,Z 154.403,A -85,B 0,C 180,E1 -8564.052,E2 -8564.052} C_VEL
LIN {X 0,Y 446.491,Z 153.208,A -85,B 0,C 180,E1 -8564.212,E2 -8564.212} C_VEL
LIN {X 0,Y 446.978,Z 140.194,A -85,B 0,C 180,E1 -8567.382,E2 -8567.382} C_VEL
LIN {X 0,Y 447.139,Z 132.011,A -85,B 0,C 180,E1 -8569.427,E2 -8569.427} C_VEL
LIN {X 0,Y 446.525,Z 127.792,A -85,B 0,C 180,E1 -8570.559,E2 -8570.559} C_VEL
LIN {X 0,Y 446.464,Z 127.685,A -85,B 0,C 180,E1 -8574.159,E2 -8574.159} C_VEL
LIN {X 0,Y 446.473,Z 127.679,A -85,B 0,C 180,E1 -8577.161,E2 -8577.161} C_VEL
LIN {X 0,Y 446.428,Z 127.692,A -85,B 0,C 180,E1 -8580.249,E2 -8580.249} C_VEL
LIN {X 0,Y 446.445,Z 127.683,A -85,B 0,C 180,E1 -8583.453,E2 -8583.453} C_VEL
LIN {X 0,Y 446.402,Z 127.688,A -85,B 0,C 180,E1 -8586.745,E2 -8586.745} C_VEL
LIN {X 0,Y 446.478,Z 127.681,A -85,B 0,C 180,E1 -8589.528,E2 -8589.528} C_VEL
LIN {X 0,Y 446.428,Z 127.685,A -85,B 0,C 180,E1 -8592.604,E2 -8592.604} C_VEL
LIN {X 0,Y 446.451,Z 127.683,A -85,B 0,C 180,E1 -8595.103,E2 -8595.103} C_VEL
LIN {X 0,Y 446.427,Z 127.684,A -85,B 0,C 180,E1 -8598.609,E2 -8598.609} C_VEL
LIN {X 0,Y 446.437,Z 127.685,A -85,B 0,C 180,E1 -8600.972,E2 -8600.972} C_VEL
LIN {X 0,Y 446.42,Z 127.685,A -85,B 0,C 180,E1 -8604.374,E2 -8604.374} C_VEL
LIN {X 0,Y 446.421,Z 127.688,A -85,B 0,C 180,E1 -8607.638,E2 -8607.638} C_VEL
LIN {X 0,Y 446.447,Z 127.686,A -85,B 0,C 180,E1 -8610.79,E2 -8610.79} C_VEL
LIN {X 0,Y 446.476,Z 127.678,A -85,B 0,C 180,E1 -8613.848,E2 -8613.848} C_VEL
LIN {X 0,Y 446.428,Z 127.692,A -85,B 0,C 180,E1 -8616.823,E2 -8616.823} C_VEL
LIN {X 0,Y 446.443,Z 127.682,A -85,B 0,C 180,E1 -8619.737,E2 -8619.737} C_VEL
LIN {X 0,Y 446.463,Z 127.687,A -85,B 0,C 180,E1 -8622.597,E2 -8622.597} C_VEL
LIN {X 0,Y 446.469,Z 127.679,A -85,B 0,C 180,E1 -8625.412,E2 -8625.412} C_VEL
LIN {X 0,Y 446.538,Z 127.675,A -85,B 0,C 180,E1 -8628.194,E2 -8628.194} C_VEL
LIN {X 0,Y 446.599,Z 127.666,A -85,B 0,C 180,E1 -8631.858,E2 -8631.858} C_VEL
LIN {X 0,Y 446.644,Z 127.66,A -85,B 0,C 180,E1 -8634.582,E2 -8634.582} C_VEL
LIN {X 0,Y 446.707,Z 127.65,A -85,B 0,C 180,E1 -8637.295,E2 -8637.295} C_VEL
LIN {X 0,Y 446.793,Z 127.646,A -85,B 0,C 180,E1 -8640,E2 -8640} C_VEL
LIN {X 0,Y 446.69,Z 127.652,A -85,B 0,C 180,E1 -8642.705,E2 -8642.705} C_VEL
LIN {X 0,Y 446.645,Z 127.659,A -85,B 0,C 180,E1 -8646.324,E2 -8646.324} C_VEL
LIN {X 0,Y 446.536,Z 127.672,A -85,B 0,C 180,E1 -8649.055,E2 -8649.055} C_VEL
LIN {X 0,Y 446.52,Z 127.673,A -85,B 0,C 180,E1 -8652.73,E2 -8652.73} C_VEL
LIN {X 0,Y 446.494,Z 127.676,A -85,B 0,C 180,E1 -8656.228,E2 -8656.228} C_VEL
LIN {X 0,Y 446.468,Z 127.686,A -85,B 0,C 180,E1 -8659.303,E2 -8659.303} C_VEL
LIN {X 0,Y 446.416,Z 127.686,A -85,B 0,C 180,E1 -8662.2,E2 -8662.2} C_VEL
LIN {X 0,Y 446.456,Z 127.687,A -85,B 0,C 180,E1 -8665.152,E2 -8665.152} C_VEL
LIN {X 0,Y 446.483,Z 127.678,A -85,B 0,C 180,E1 -8668.179,E2 -8668.179} C_VEL
LIN {X 0,Y 446.417,Z 127.686,A -85,B 0,C 180,E1 -8671.775,E2 -8671.775} C_VEL
LIN {X 0,Y 446.429,Z 127.69,A -85,B 0,C 180,E1 -8674.523,E2 -8674.523} C_VEL
LIN {X 0,Y 446.412,Z 127.689,A -85,B 0,C 180,E1 -8678.079,E2 -8678.079} C_VEL
LIN {X 0,Y 446.424,Z 127.687,A -85,B 0,C 180,E1 -8680.918,E2 -8680.918} C_VEL
LIN {X 0,Y 446.398,Z 127.69,A -85,B 0,C 180,E1 -8683.846,E2 -8683.846} C_VEL
LIN {X 0,Y 446.396,Z 127.693,A -85,B 0,C 180,E1 -8686.404,E2 -8686.404} C_VEL
LIN {X 0,Y 446.425,Z 127.685,A -85,B 0,C 180,E1 -8689.083,E2 -8689.083} C_VEL
LIN {X 0,Y 446.408,Z 127.693,A -85,B 0,C 180,E1 -8692.122,E2 -8692.122} C_VEL
LIN {X 0,Y 446.428,Z 127.687,A -85,B 0,C 180,E1 -8695.477,E2 -8695.477} C_VEL
LIN {X 0,Y 446.414,Z 127.686,A -85,B 0,C 180,E1 -8698.7,E2 -8698.7} C_VEL
LIN {X 0,Y 446.484,Z 127.682,A -85,B 0,C 180,E1 -8701.822,E2 -8701.822} C_VEL
LIN {X 0,Y 446.457,Z 127.675,A -85,B 0,C 180,E1 -8704.848,E2 -8704.848} C_VEL
LIN {X 0,Y 446.493,Z 127.786,A -85,B 0,C 180,E1 -8706.582,E2 -8706.582} C_VEL
LIN {X 0,Y 447.697,Z 135.166,A -85,B 0,C 180,E1 -8708.385,E2 -8708.385} C_VEL
LIN {X 0,Y 447.366,Z 145.546,A -85,B 0,C 180,E1 -8710.737,E2 -8710.737} C_VEL
LIN {X 0,Y 446.677,Z 160.462,A -85,B 0,C 180,E1 -8714.069,E2 -8714.069} C_VEL
LIN {X 0,Y 446.396,Z 169.183,A -85,B 0,C 180,E1 -8715.948,E2 -8715.948} C_VEL
LIN {X 0,Y 447.281,Z 175.543,A -85,B 0,C 180,E1 -8716.118,E2 -8716.118} C_VEL
LIN {X 0,Y 448.78,Z 187.817,A -85,B 0,C 180,E1 -8716.363,E2 -8716.363} C_VEL
LIN {X 0,Y 448.473,Z 245.698,A -85,B 0,C 180,E1 -8717.31,E2 -8717.31} C_VEL
LIN {X 0,Y 448.161,Z 255.241,A -85,B 0,C 180,E1 -8717.577,E2 -8717.577} C_VEL
LIN {X 0,Y 447.846,Z 265.29,A -85,B 0,C 180,E1 -8717.999,E2 -8717.999} C_VEL
LIN {X 0,Y 447.468,Z 276.703,A -85,B 0,C 180,E1 -8718.678,E2 -8718.678} C_VEL
LIN {X 0,Y 447.066,Z 285.289,A -85,B 0,C 180,E1 -8719.356,E2 -8719.356} C_VEL
LIN {X 0,Y 446.635,Z 293.366,A -85,B 0,C 180,E1 -8720.147,E2 -8720.147} C_VEL
LIN {X 0,Y 446.348,Z 300.04,A -85,B 0,C 180,E1 -8720.941,E2 -8720.941} C_VEL
LIN {X 0,Y 446.058,Z 306.374,A -85,B 0,C 180,E1 -8721.848,E2 -8721.848} C_VEL
LIN {X 0,Y 445.821,Z 311.638,A -85,B 0,C 180,E1 -8722.755,E2 -8722.755} C_VEL
LIN {X 0,Y 445.664,Z 316.027,A -85,B 0,C 180,E1 -8723.663,E2 -8723.663} C_VEL
LIN {X 0,Y 445.516,Z 321.203,A -85,B 0,C 180,E1 -8725.023,E2 -8725.023} C_VEL
LIN {X 0,Y 445.417,Z 325.002,A -85,B 0,C 180,E1 -8726.382,E2 -8726.382} C_VEL
LIN {X 0,Y 445.411,Z 326.75,A -85,B 0,C 180,E1 -8727.287,E2 -8727.287} C_VEL
LIN {X 0,Y 445.351,Z 328,A -85,B 0,C 180,E1 -8728.192,E2 -8728.192} C_VEL
LIN {X 0,Y 445.313,Z 328.779,A -85,B 0,C 180,E1 -8729.096,E2 -8729.096} C_VEL
LIN {X 0,Y 445.315,Z 329.074,A -85,B 0,C 180,E1 -8730,E2 -8730} C_VEL
LIN {X 0,Y 445.313,Z 328.777,A -85,B 0,C 180,E1 -8730.905,E2 -8730.905} C_VEL
LIN {X 0,Y 445.351,Z 327.995,A -85,B 0,C 180,E1 -8731.809,E2 -8731.809} C_VEL
LIN {X 0,Y 445.411,Z 326.741,A -85,B 0,C 180,E1 -8732.713,E2 -8732.713} C_VEL
LIN {X 0,Y 445.412,Z 323.836,A -85,B 0,C 180,E1 -8734.072,E2 -8734.072} C_VEL
LIN {X 0,Y 445.516,Z 321.189,A -85,B 0,C 180,E1 -8734.978,E2 -8734.978} C_VEL
LIN {X 0,Y 445.664,Z 316.007,A -85,B 0,C 180,E1 -8736.338,E2 -8736.338} C_VEL
LIN {X 0,Y 445.871,Z 309.179,A -85,B 0,C 180,E1 -8737.7,E2 -8737.7} C_VEL
LIN {X 0,Y 446.266,Z 301.717,A -85,B 0,C 180,E1 -8738.833,E2 -8738.833} C_VEL
LIN {X 0,Y 446.575,Z 294.355,A -85,B 0,C 180,E1 -8739.74,E2 -8739.74} C_VEL
LIN {X 0,Y 447.014,Z 286.475,A -85,B 0,C 180,E1 -8740.531,E2 -8740.531} C_VEL
LIN {X 0,Y 447.347,Z 278.145,A -85,B 0,C 180,E1 -8741.211,E2 -8741.211} C_VEL
LIN {X 0,Y 447.803,Z 267.511,A -85,B 0,C 180,E1 -8741.888,E2 -8741.888} C_VEL
LIN {X 0,Y 448.125,Z 255.94,A -85,B 0,C 180,E1 -8742.396,E2 -8742.396} C_VEL
LIN {X 0,Y 448.394,Z 246.26,A -85,B 0,C 180,E1 -8742.676,E2 -8742.676} C_VEL
LIN {X 0,Y 448.767,Z 186.664,A -85,B 0,C 180,E1 -8743.652,E2 -8743.652} C_VEL
LIN {X 0,Y 446.398,Z 169.401,A -85,B 0,C 180,E1 -8744.028,E2 -8744.028} C_VEL
LIN {X 0,Y 446.481,Z 166.496,A -85,B 0,C 180,E1 -8744.587,E2 -8744.587} C_VEL
LIN {X 0,Y 447.045,Z 151.818,A -85,B 0,C 180,E1 -8747.852,E2 -8747.852} C_VEL
LIN {X 0,Y 447.691,Z 138.158,A -85,B 0,C 180,E1 -8750.925,E2 -8750.925} C_VEL
LIN {X 0,Y 447.452,Z 133.191,A -85,B 0,C 180,E1 -8752.075,E2 -8752.075} C_VEL
LIN {X 0,Y 446.494,Z 127.773,A -85,B 0,C 180,E1 -8753.419,E2 -8753.419} C_VEL
LIN {X 0,Y 446.476,Z 127.684,A -85,B 0,C 180,E1 -8756.203,E2 -8756.203} C_VEL
LIN {X 0,Y 446.449,Z 127.682,A -85,B 0,C 180,E1 -8759.209,E2 -8759.209} C_VEL
LIN {X 0,Y 446.423,Z 127.691,A -85,B 0,C 180,E1 -8762.362,E2 -8762.362} C_VEL
LIN {X 0,Y 446.42,Z 127.687,A -85,B 0,C 180,E1 -8765.626,E2 -8765.626} C_VEL
LIN {X 0,Y 446.444,Z 127.682,A -85,B 0,C 180,E1 -8769.027,E2 -8769.027} C_VEL
LIN {X 0,Y 446.434,Z 127.686,A -85,B 0,C 180,E1 -8772.277,E2 -8772.277} C_VEL
LIN {X 0,Y 446.451,Z 127.682,A -85,B 0,C 180,E1 -8775.104,E2 -8775.104} C_VEL
LIN {X 0,Y 446.428,Z 127.684,A -85,B 0,C 180,E1 -8778.609,E2 -8778.609} C_VEL
LIN {X 0,Y 446.439,Z 127.684,A -85,B 0,C 180,E1 -8780.973,E2 -8780.973} C_VEL
LIN {X 0,Y 446.422,Z 127.685,A -85,B 0,C 180,E1 -8784.374,E2 -8784.374} C_VEL
LIN {X 0,Y 446.423,Z 127.688,A -85,B 0,C 180,E1 -8787.639,E2 -8787.639} C_VEL
LIN {X 0,Y 446.449,Z 127.685,A -85,B 0,C 180,E1 -8790.791,E2 -8790.791} C_VEL
LIN {X 0,Y 446.479,Z 127.678,A -85,B 0,C 180,E1 -8793.849,E2 -8793.849} C_VEL
LIN {X 0,Y 446.43,Z 127.69,A -85,B 0,C 180,E1 -8796.823,E2 -8796.823} C_VEL
LIN {X 0,Y 446.445,Z 127.682,A -85,B 0,C 180,E1 -8799.737,E2 -8799.737} C_VEL
LIN {X 0,Y 446.465,Z 127.686,A -85,B 0,C 180,E1 -8802.597,E2 -8802.597} C_VEL
LIN {X 0,Y 446.471,Z 127.679,A -85,B 0,C 180,E1 -8805.413,E2 -8805.413} C_VEL
LIN {X 0,Y 446.519,Z 127.677,A -85,B 0,C 180,E1 -8808.193,E2 -8808.193} C_VEL
LIN {X 0,Y 446.602,Z 127.664,A -85,B 0,C 180,E1 -8811.858,E2 -8811.858} C_VEL
LIN {X 0,Y 446.644,Z 127.661,A -85,B 0,C 180,E1 -8814.583,E2 -8814.583} C_VEL
LIN {X 0,Y 446.666,Z 127.662,A -85,B 0,C 180,E1 -8818.197,E2 -8818.197} C_VEL
LIN {X 0,Y 446.794,Z 127.646,A -85,B 0,C 180,E1 -8820,E2 -8820} C_VEL
LIN {X 0,Y 446.692,Z 127.652,A -85,B 0,C 180,E1 -8822.705,E2 -8822.705} C_VEL
LIN {X 0,Y 446.648,Z 127.659,A -85,B 0,C 180,E1 -8826.324,E2 -8826.324} C_VEL
LIN {X 0,Y 446.54,Z 127.671,A -85,B 0,C 180,E1 -8829.055,E2 -8829.055} C_VEL
LIN {X 0,Y 446.536,Z 127.671,A -85,B 0,C 180,E1 -8832.729,E2 -8832.729} C_VEL
LIN {X 0,Y 446.492,Z 127.676,A -85,B 0,C 180,E1 -8836.459,E2 -8836.459} C_VEL
LIN {X 0,Y 446.471,Z 127.686,A -85,B 0,C 180,E1 -8839.303,E2 -8839.303} C_VEL
LIN {X 0,Y 446.419,Z 127.685,A -85,B 0,C 180,E1 -8842.2,E2 -8842.2} C_VEL
LIN {X 0,Y 446.459,Z 127.688,A -85,B 0,C 180,E1 -8845.152,E2 -8845.152} C_VEL
LIN {X 0,Y 446.486,Z 127.677,A -85,B 0,C 180,E1 -8848.179,E2 -8848.179} C_VEL
LIN {X 0,Y 446.421,Z 127.685,A -85,B 0,C 180,E1 -8851.775,E2 -8851.775} C_VEL
LIN {X 0,Y 446.432,Z 127.688,A -85,B 0,C 180,E1 -8854.523,E2 -8854.523} C_VEL
LIN {X 0,Y 446.415,Z 127.687,A -85,B 0,C 180,E1 -8858.079,E2 -8858.079} C_VEL
LIN {X 0,Y 446.428,Z 127.687,A -85,B 0,C 180,E1 -8860.918,E2 -8860.918} C_VEL
LIN {X 0,Y 446.399,Z 127.689,A -85,B 0,C 180,E1 -8863.846,E2 -8863.846} C_VEL
LIN {X 0,Y 446.4,Z 127.695,A -85,B 0,C 180,E1 -8866.403,E2 -8866.403} C_VEL
LIN {X 0,Y 446.428,Z 127.684,A -85,B 0,C 180,E1 -8869.082,E2 -8869.082} C_VEL
LIN {X 0,Y 446.432,Z 127.689,A -85,B 0,C 180,E1 -8871.918,E2 -8871.918} C_VEL
LIN {X 0,Y 446.431,Z 127.686,A -85,B 0,C 180,E1 -8875.477,E2 -8875.477} C_VEL
LIN {X 0,Y 446.417,Z 127.686,A -85,B 0,C 180,E1 -8878.7,E2 -8878.7} C_VEL
LIN {X 0,Y 446.487,Z 127.684,A -85,B 0,C 180,E1 -8881.821,E2 -8881.821} C_VEL
LIN {X 0,Y 446.446,Z 127.682,A -85,B 0,C 180,E1 -8884.847,E2 -8884.847} C_VEL
LIN {X 0,Y 446.45,Z 127.687,A -85,B 0,C 180,E1 -8888.245,E2 -8888.245} C_VEL
LIN {X 0,Y 446.539,Z 127.837,A -85,B 0,C 180,E1 -8889.561,E2 -8889.561} C_VEL
LIN {X 0,Y 447.152,Z 132.234,A -85,B 0,C 180,E1 -8890.727,E2 -8890.727} C_VEL
LIN {X 0,Y 446.889,Z 141.705,A -85,B 0,C 180,E1 -8893.086,E2 -8893.086} C_VEL
LIN {X 0,Y 446.52,Z 153.674,A -85,B 0,C 180,E1 -8895.976,E2 -8895.976} C_VEL
LIN {X 0,Y 446.732,Z 155.399,A -85,B 0,C 180,E1 -8896.078,E2 -8896.078} C_VEL
LIN {X 0,Y 448.889,Z 168.914,A -85,B 0,C 180,E1 -8896.365,E2 -8896.365} C_VEL
LIN {X 0,Y 448.637,Z 211.646,A -85,B 0,C 180,E1 -8897.046,E2 -8897.046} C_VEL
LIN {X 0,Y 447.805,Z 217.487,A -85,B 0,C 180,E1 -8897.111,E2 -8897.111} C_VEL
LIN {X 0,Y 442.228,Z 234.925,A -85,B 0,C 180,E1 -8897.296,E2 -8897.296} C_VEL
LIN {X 0,Y 441.412,Z 240.144,A -85,B 0,C 180,E1 -8897.453,E2 -8897.453} C_VEL
LIN {X 0,Y 441.322,Z 242.049,A -85,B 0,C 180,E1 -8897.519,E2 -8897.519} C_VEL
LIN {X 0,Y 440.938,Z 252.963,A -85,B 0,C 180,E1 -8898.041,E2 -8898.041} C_VEL
LIN {X 0,Y 440.631,Z 263.305,A -85,B 0,C 180,E1 -8898.733,E2 -8898.733} C_VEL
LIN {X 0,Y 440.247,Z 270.218,A -85,B 0,C 180,E1 -8899.305,E2 -8899.305} C_VEL
LIN {X 0,Y 439.926,Z 278.153,A -85,B 0,C 180,E1 -8900.111,E2 -8900.111} C_VEL
LIN {X 0,Y 439.572,Z 283.855,A -85,B 0,C 180,E1 -8900.8,E2 -8900.8} C_VEL
LIN {X 0,Y 439.2,Z 290.217,A -85,B 0,C 180,E1 -8901.719,E2 -8901.719} C_VEL
LIN {X 0,Y 438.977,Z 296.638,A -85,B 0,C 180,E1 -8902.866,E2 -8902.866} C_VEL
LIN {X 0,Y 438.755,Z 301.823,A -85,B 0,C 180,E1 -8904.023,E2 -8904.023} C_VEL
LIN {X 0,Y 438.472,Z 306.595,A -85,B 0,C 180,E1 -8905.403,E2 -8905.403} C_VEL
LIN {X 0,Y 438.451,Z 308.919,A -85,B 0,C 180,E1 -8906.324,E2 -8906.324} C_VEL
LIN {X 0,Y 438.391,Z 310.69,A -85,B 0,C 180,E1 -8907.243,E2 -8907.243} C_VEL
LIN {X 0,Y 438.281,Z 311.969,A -85,B 0,C 180,E1 -8908.162,E2 -8908.162} C_VEL
LIN {X 0,Y 438.23,Z 312.778,A -85,B 0,C 180,E1 -8909.081,E2 -8909.081} C_VEL
LIN {X 0,Y 438.228,Z 313.086,A -85,B 0,C 180,E1 -8910,E2 -8910} C_VEL
LIN {X 0,Y 438.23,Z 312.811,A -85,B 0,C 180,E1 -8910.919,E2 -8910.919} C_VEL
LIN {X 0,Y 438.281,Z 312.069,A -85,B 0,C 180,E1 -8911.838,E2 -8911.838} C_VEL
LIN {X 0,Y 438.39,Z 310.858,A -85,B 0,C 180,E1 -8912.756,E2 -8912.756} C_VEL
LIN {X 0,Y 438.463,Z 308.01,A -85,B 0,C 180,E1 -8914.136,E2 -8914.136} C_VEL
LIN {X 0,Y 438.532,Z 305.419,A -85,B 0,C 180,E1 -8915.057,E2 -8915.057} C_VEL
LIN {X 0,Y 438.846,Z 300.311,A -85,B 0,C 180,E1 -8916.436,E2 -8916.436} C_VEL
LIN {X 0,Y 439.012,Z 294.82,A -85,B 0,C 180,E1 -8917.589,E2 -8917.589} C_VEL
LIN {X 0,Y 439.36,Z 287.924,A -85,B 0,C 180,E1 -8918.74,E2 -8918.74} C_VEL
LIN {X 0,Y 439.811,Z 280.002,A -85,B 0,C 180,E1 -8919.775,E2 -8919.775} C_VEL
LIN {X 0,Y 440.161,Z 272.448,A -85,B 0,C 180,E1 -8920.58,E2 -8920.58} C_VEL
LIN {X 0,Y 440.496,Z 264.533,A -85,B 0,C 180,E1 -8921.27,E2 -8921.27} C_VEL
LIN {X 0,Y 440.895,Z 256.36,A -85,B 0,C 180,E1 -8921.843,E2 -8921.843} C_VEL
LIN {X 0,Y 441.194,Z 248.086,A -85,B 0,C 180,E1 -8922.301,E2 -8922.301} C_VEL
LIN {X 0,Y 441.456,Z 239.158,A -85,B 0,C 180,E1 -8922.673,E2 -8922.673} C_VEL
LIN {X 0,Y 441.653,Z 230.366,A -85,B 0,C 180,E1 -8922.927,E2 -8922.927} C_VEL
LIN {X 0,Y 441.948,Z 168.783,A -85,B 0,C 180,E1 -8923.954,E2 -8923.954} C_VEL
LIN {X 0,Y 439.53,Z 154.408,A -85,B 0,C 180,E1 -8924.29,E2 -8924.29} C_VEL
LIN {X 0,Y 439.514,Z 153.214,A -85,B 0,C 180,E1 -8924.468,E2 -8924.468} C_VEL
LIN {X 0,Y 439.998,Z 140.283,A -85,B 0,C 180,E1 -8927.667,E2 -8927.667} C_VEL
LIN {X 0,Y 440.084,Z 132.695,A -85,B 0,C 180,E1 -8929.594,E2 -8929.594} C_VEL
LIN {X 0,Y 439.453,Z 128.657,A -85,B 0,C 180,E1 -8930.722,E2 -8930.722} C_VEL
LIN {X 0,Y 439.411,Z 128.565,A -85,B 0,C 180,E1 -8934.572,E2 -8934.572} C_VEL
LIN {X 0,Y 439.441,Z 128.555,A -85,B 0,C 180,E1 -8937.632,E2 -8937.632} C_VEL
LIN {X 0,Y 439.361,Z 128.566,A -85,B 0,C 180,E1 -8940.788,E2 -8940.788} C_VEL
LIN {X 0,Y 439.387,Z 128.568,A -85,B 0,C 180,E1 -8944.043,E2 -8944.043} C_VEL
LIN {X 0,Y 439.351,Z 128.566,A -85,B 0,C 180,E1 -8946.887,E2 -8946.887} C_VEL
LIN {X 0,Y 439.413,Z 128.565,A -85,B 0,C 180,E1 -8949.851,E2 -8949.851} C_VEL
LIN {X 0,Y 439.381,Z 128.562,A -85,B 0,C 180,E1 -8952.627,E2 -8952.627} C_VEL
LIN {X 0,Y 439.399,Z 128.563,A -85,B 0,C 180,E1 -8955.27,E2 -8955.27} C_VEL
LIN {X 0,Y 439.387,Z 128.562,A -85,B 0,C 180,E1 -8958.743,E2 -8958.743} C_VEL
LIN {X 0,Y 439.371,Z 128.569,A -85,B 0,C 180,E1 -8961.608,E2 -8961.608} C_VEL
LIN {X 0,Y 439.4,Z 128.562,A -85,B 0,C 180,E1 -8964.844,E2 -8964.844} C_VEL
LIN {X 0,Y 439.372,Z 128.563,A -85,B 0,C 180,E1 -8968.139,E2 -8968.139} C_VEL
LIN {X 0,Y 439.431,Z 128.558,A -85,B 0,C 180,E1 -8971.598,E2 -8971.598} C_VEL
LIN {X 0,Y 439.404,Z 128.561,A -85,B 0,C 180,E1 -8974.415,E2 -8974.415} C_VEL
LIN {X 0,Y 439.364,Z 128.566,A -85,B 0,C 180,E1 -8977.424,E2 -8977.424} C_VEL
LIN {X 0,Y 439.44,Z 128.562,A -85,B 0,C 180,E1 -8980.662,E2 -8980.662} C_VEL
LIN {X 0,Y 439.461,Z 128.555,A -85,B 0,C 180,E1 -8984.224,E2 -8984.224} C_VEL
LIN {X 0,Y 439.506,Z 128.549,A -85,B 0,C 180,E1 -8988.002,E2 -8988.002} C_VEL
LIN {X 0,Y 439.547,Z 128.543,A -85,B 0,C 180,E1 -8991.726,E2 -8991.726} C_VEL
LIN {X 0,Y 439.62,Z 128.536,A -85,B 0,C 180,E1 -8994.496,E2 -8994.496} C_VEL
LIN {X 0,Y 439.634,Z 128.537,A -85,B 0,C 180,E1 -8998.168,E2 -8998.168} C_VEL
LIN {X 0,Y 439.763,Z 128.522,A -85,B 0,C 180,E1 -9000,E2 -9000} C_VEL
LIN {X 0,Y 439.639,Z 128.53,A -85,B 0,C 180,E1 -9002.749,E2 -9002.749} C_VEL
LIN {X 0,Y 439.617,Z 128.534,A -85,B 0,C 180,E1 -9006.425,E2 -9006.425} C_VEL
LIN {X 0,Y 439.498,Z 128.55,A -85,B 0,C 180,E1 -9009.202,E2 -9009.202} C_VEL
LIN {X 0,Y 439.464,Z 128.554,A -85,B 0,C 180,E1 -9012.938,E2 -9012.938} C_VEL
LIN {X 0,Y 439.446,Z 128.554,A -85,B 0,C 180,E1 -9016.349,E2 -9016.349} C_VEL
LIN {X 0,Y 439.401,Z 128.563,A -85,B 0,C 180,E1 -9019.626,E2 -9019.626} C_VEL
LIN {X 0,Y 439.363,Z 128.566,A -85,B 0,C 180,E1 -9022.575,E2 -9022.575} C_VEL
LIN {X 0,Y 439.403,Z 128.561,A -85,B 0,C 180,E1 -9025.585,E2 -9025.585} C_VEL
LIN {X 0,Y 439.415,Z 128.563,A -85,B 0,C 180,E1 -9028.673,E2 -9028.673} C_VEL
LIN {X 0,Y 439.368,Z 128.564,A -85,B 0,C 180,E1 -9032.03,E2 -9032.03} C_VEL
LIN {X 0,Y 439.394,Z 128.561,A -85,B 0,C 180,E1 -9035.341,E2 -9035.341} C_VEL
LIN {X 0,Y 439.373,Z 128.569,A -85,B 0,C 180,E1 -9038.596,E2 -9038.596} C_VEL
LIN {X 0,Y 439.386,Z 128.562,A -85,B 0,C 180,E1 -9041.257,E2 -9041.257} C_VEL
LIN {X 0,Y 439.398,Z 128.562,A -85,B 0,C 180,E1 -9044.73,E2 -9044.73} C_VEL
LIN {X 0,Y 439.394,Z 128.564,A -85,B 0,C 180,E1 -9047.796,E2 -9047.796} C_VEL
LIN {X 0,Y 439.424,Z 128.562,A -85,B 0,C 180,E1 -9050.228,E2 -9050.228} C_VEL
LIN {X 0,Y 439.373,Z 128.568,A -85,B 0,C 180,E1 -9053.713,E2 -9053.713} C_VEL
LIN {X 0,Y 439.37,Z 128.564,A -85,B 0,C 180,E1 -9057.054,E2 -9057.054} C_VEL
LIN {X 0,Y 439.381,Z 128.563,A -85,B 0,C 180,E1 -9060.274,E2 -9060.274} C_VEL
LIN {X 0,Y 439.428,Z 128.562,A -85,B 0,C 180,E1 -9063.397,E2 -9063.397} C_VEL
LIN {X 0,Y 439.456,Z 128.683,A -85,B 0,C 180,E1 -9066.434,E2 -9066.434} C_VEL
LIN {X 0,Y 440.725,Z 137.005,A -85,B 0,C 180,E1 -9068.484,E2 -9068.484} C_VEL
LIN {X 0,Y 440.314,Z 147.521,A -85,B 0,C 180,E1 -9070.901,E2 -9070.901} C_VEL
LIN {X 0,Y 439.604,Z 163.25,A -85,B 0,C 180,E1 -9074.468,E2 -9074.468} C_VEL
LIN {X 0,Y 439.391,Z 168.922,A -85,B 0,C 180,E1 -9075.705,E2 -9075.705} C_VEL
LIN {X 0,Y 439.875,Z 172.85,A -85,B 0,C 180,E1 -9075.837,E2 -9075.837} C_VEL
LIN {X 0,Y 441.854,Z 187.707,A -85,B 0,C 180,E1 -9076.145,E2 -9076.145} C_VEL
LIN {X 0,Y 441.564,Z 245.616,A -85,B 0,C 180,E1 -9077.108,E2 -9077.108} C_VEL
LIN {X 0,Y 441.243,Z 255.122,A -85,B 0,C 180,E1 -9077.379,E2 -9077.379} C_VEL
LIN {X 0,Y 440.903,Z 265.168,A -85,B 0,C 180,E1 -9077.807,E2 -9077.807} C_VEL
LIN {X 0,Y 440.493,Z 276.578,A -85,B 0,C 180,E1 -9078.496,E2 -9078.496} C_VEL
LIN {X 0,Y 440.092,Z 285.164,A -85,B 0,C 180,E1 -9079.185,E2 -9079.185} C_VEL
LIN {X 0,Y 439.63,Z 293.24,A -85,B 0,C 180,E1 -9079.989,E2 -9079.989} C_VEL
LIN {X 0,Y 439.328,Z 299.913,A -85,B 0,C 180,E1 -9080.795,E2 -9080.795} C_VEL
LIN {X 0,Y 439.013,Z 306.247,A -85,B 0,C 180,E1 -9081.716,E2 -9081.716} C_VEL
LIN {X 0,Y 438.78,Z 311.511,A -85,B 0,C 180,E1 -9082.638,E2 -9082.638} C_VEL
LIN {X 0,Y 438.591,Z 315.9,A -85,B 0,C 180,E1 -9083.56,E2 -9083.56} C_VEL
LIN {X 0,Y 438.45,Z 321.075,A -85,B 0,C 180,E1 -9084.942,E2 -9084.942} C_VEL
LIN {X 0,Y 438.316,Z 324.874,A -85,B 0,C 180,E1 -9086.323,E2 -9086.323} C_VEL
LIN {X 0,Y 438.309,Z 326.621,A -85,B 0,C 180,E1 -9087.243,E2 -9087.243} C_VEL
LIN {X 0,Y 438.273,Z 327.872,A -85,B 0,C 180,E1 -9088.162,E2 -9088.162} C_VEL
LIN {X 0,Y 438.228,Z 328.651,A -85,B 0,C 180,E1 -9089.081,E2 -9089.081} C_VEL
LIN {X 0,Y 438.227,Z 328.945,A -85,B 0,C 180,E1 -9090,E2 -9090} C_VEL
LIN {X 0,Y 438.228,Z 328.649,A -85,B 0,C 180,E1 -9090.919,E2 -9090.919} C_VEL
LIN {X 0,Y 438.273,Z 327.867,A -85,B 0,C 180,E1 -9091.838,E2 -9091.838} C_VEL
LIN {X 0,Y 438.309,Z 326.612,A -85,B 0,C 180,E1 -9092.757,E2 -9092.757} C_VEL
LIN {X 0,Y 438.324,Z 323.706,A -85,B 0,C 180,E1 -9094.138,E2 -9094.138} C_VEL
LIN {X 0,Y 438.45,Z 321.059,A -85,B 0,C 180,E1 -9095.058,E2 -9095.058} C_VEL
LIN {X 0,Y 438.613,Z 315.348,A -85,B 0,C 180,E1 -9096.567,E2 -9096.567} C_VEL
LIN {X 0,Y 438.827,Z 309.049,A -85,B 0,C 180,E1 -9097.824,E2 -9097.824} C_VEL
LIN {X 0,Y 439.248,Z 301.586,A -85,B 0,C 180,E1 -9098.975,E2 -9098.975} C_VEL
LIN {X 0,Y 439.584,Z 294.224,A -85,B 0,C 180,E1 -9099.897,E2 -9099.897} C_VEL
LIN {X 0,Y 440.039,Z 286.343,A -85,B 0,C 180,E1 -9100.7,E2 -9100.7} C_VEL
LIN {X 0,Y 440.393,Z 278.013,A -85,B 0,C 180,E1 -9101.39,E2 -9101.39} C_VEL
LIN {X 0,Y 440.866,Z 267.377,A -85,B 0,C 180,E1 -9102.077,E2 -9102.077} C_VEL
LIN {X 0,Y 441.211,Z 255.804,A -85,B 0,C 180,E1 -9102.593,E2 -9102.593} C_VEL
LIN {X 0,Y 441.482,Z 246.119,A -85,B 0,C 180,E1 -9102.878,E2 -9102.878} C_VEL
LIN {X 0,Y 441.893,Z 187.686,A -85,B 0,C 180,E1 -9103.85,E2 -9103.85} C_VEL
LIN {X 0,Y 439.411,Z 169.391,A -85,B 0,C 180,E1 -9104.248,E2 -9104.248} C_VEL
LIN {X 0,Y 439.423,Z 167.519,A -85,B 0,C 180,E1 -9104.567,E2 -9104.567} C_VEL
LIN {X 0,Y 440.012,Z 152.739,A -85,B 0,C 180,E1 -9107.907,E2 -9107.907} C_VEL
LIN {X 0,Y 440.676,Z 140.137,A -85,B 0,C 180,E1 -9110.784,E2 -9110.784} C_VEL
LIN {X 0,Y 440.599,Z 135.469,A -85,B 0,C 180,E1 -9111.874,E2 -9111.874} C_VEL
LIN {X 0,Y 439.455,Z 128.67,A -85,B 0,C 180,E1 -9113.567,E2 -9113.567} C_VEL
LIN {X 0,Y 439.429,Z 128.562,A -85,B 0,C 180,E1 -9116.604,E2 -9116.604} C_VEL
LIN {X 0,Y 439.383,Z 128.563,A -85,B 0,C 180,E1 -9119.726,E2 -9119.726} C_VEL
LIN {X 0,Y 439.373,Z 128.564,A -85,B 0,C 180,E1 -9122.946,E2 -9122.946} C_VEL
LIN {X 0,Y 439.374,Z 128.568,A -85,B 0,C 180,E1 -9126.287,E2 -9126.287} C_VEL
LIN {X 0,Y 439.402,Z 128.566,A -85,B 0,C 180,E1 -9129.849,E2 -9129.849} C_VEL
LIN {X 0,Y 439.381,Z 128.563,A -85,B 0,C 180,E1 -9132.627,E2 -9132.627} C_VEL
LIN {X 0,Y 439.399,Z 128.562,A -85,B 0,C 180,E1 -9135.271,E2 -9135.271} C_VEL
LIN {X 0,Y 439.389,Z 128.561,A -85,B 0,C 180,E1 -9138.743,E2 -9138.743} C_VEL
LIN {X 0,Y 439.373,Z 128.57,A -85,B 0,C 180,E1 -9141.608,E2 -9141.608} C_VEL
LIN {X 0,Y 439.401,Z 128.561,A -85,B 0,C 180,E1 -9144.844,E2 -9144.844} C_VEL
LIN {X 0,Y 439.374,Z 128.563,A -85,B 0,C 180,E1 -9148.14,E2 -9148.14} C_VEL
LIN {X 0,Y 439.433,Z 128.558,A -85,B 0,C 180,E1 -9151.598,E2 -9151.598} C_VEL
LIN {X 0,Y 439.406,Z 128.56,A -85,B 0,C 180,E1 -9154.415,E2 -9154.415} C_VEL
LIN {X 0,Y 439.366,Z 128.566,A -85,B 0,C 180,E1 -9157.425,E2 -9157.425} C_VEL
LIN {X 0,Y 439.443,Z 128.56,A -85,B 0,C 180,E1 -9160.663,E2 -9160.663} C_VEL
LIN {X 0,Y 439.464,Z 128.554,A -85,B 0,C 180,E1 -9164.225,E2 -9164.225} C_VEL
LIN {X 0,Y 439.485,Z 128.551,A -85,B 0,C 180,E1 -9168.001,E2 -9168.001} C_VEL
LIN {X 0,Y 439.55,Z 128.542,A -85,B 0,C 180,E1 -9171.726,E2 -9171.726} C_VEL
LIN {X 0,Y 439.619,Z 128.537,A -85,B 0,C 180,E1 -9174.496,E2 -9174.496} C_VEL
LIN {X 0,Y 439.636,Z 128.538,A -85,B 0,C 180,E1 -9178.168,E2 -9178.168} C_VEL
LIN {X 0,Y 439.764,Z 128.521,A -85,B 0,C 180,E1 -9180,E2 -9180} C_VEL
LIN {X 0,Y 439.641,Z 128.53,A -85,B 0,C 180,E1 -9182.749,E2 -9182.749} C_VEL
LIN {X 0,Y 439.62,Z 128.534,A -85,B 0,C 180,E1 -9186.425,E2 -9186.425} C_VEL
LIN {X 0,Y 439.502,Z 128.549,A -85,B 0,C 180,E1 -9189.202,E2 -9189.202} C_VEL
LIN {X 0,Y 439.506,Z 128.547,A -85,B 0,C 180,E1 -9192.727,E2 -9192.727} C_VEL
LIN {X 0,Y 439.449,Z 128.554,A -85,B 0,C 180,E1 -9196.349,E2 -9196.349} C_VEL
LIN {X 0,Y 439.404,Z 128.563,A -85,B 0,C 180,E1 -9199.626,E2 -9199.626} C_VEL
LIN {X 0,Y 439.366,Z 128.565,A -85,B 0,C 180,E1 -9202.575,E2 -9202.575} C_VEL
LIN {X 0,Y 439.407,Z 128.561,A -85,B 0,C 180,E1 -9205.585,E2 -9205.585} C_VEL
LIN {X 0,Y 439.419,Z 128.561,A -85,B 0,C 180,E1 -9208.673,E2 -9208.673} C_VEL
LIN {X 0,Y 439.372,Z 128.564,A -85,B 0,C 180,E1 -9212.03,E2 -9212.03} C_VEL
LIN {X 0,Y 439.398,Z 128.561,A -85,B 0,C 180,E1 -9215.341,E2 -9215.341} C_VEL
LIN {X 0,Y 439.377,Z 128.57,A -85,B 0,C 180,E1 -9218.596,E2 -9218.596} C_VEL
LIN {X 0,Y 439.39,Z 128.562,A -85,B 0,C 180,E1 -9221.257,E2 -9221.257} C_VEL
LIN {X 0,Y 439.4,Z 128.563,A -85,B 0,C 180,E1 -9224.73,E2 -9224.73} C_VEL
LIN {X 0,Y 439.397,Z 128.562,A -85,B 0,C 180,E1 -9227.796,E2 -9227.796} C_VEL
LIN {X 0,Y 439.438,Z 128.562,A -85,B 0,C 180,E1 -9230.228,E2 -9230.228} C_VEL
LIN {X 0,Y 439.378,Z 128.566,A -85,B 0,C 180,E1 -9233.713,E2 -9233.713} C_VEL
LIN {X 0,Y 439.374,Z 128.563,A -85,B 0,C 180,E1 -9237.054,E2 -9237.054} C_VEL
LIN {X 0,Y 439.384,Z 128.564,A -85,B 0,C 180,E1 -9240.274,E2 -9240.274} C_VEL
LIN {X 0,Y 439.43,Z 128.56,A -85,B 0,C 180,E1 -9243.396,E2 -9243.396} C_VEL
LIN {X 0,Y 439.386,Z 128.565,A -85,B 0,C 180,E1 -9246.429,E2 -9246.429} C_VEL
LIN {X 0,Y 439.485,Z 128.805,A -85,B 0,C 180,E1 -9249.463,E2 -9249.463} C_VEL
LIN {X 0,Y 440.174,Z 134.259,A -85,B 0,C 180,E1 -9250.908,E2 -9250.908} C_VEL
LIN {X 0,Y 439.757,Z 146.042,A -85,B 0,C 180,E1 -9253.864,E2 -9253.864} C_VEL
LIN {X 0,Y 439.51,Z 153.867,A -85,B 0,C 180,E1 -9255.755,E2 -9255.755} C_VEL
LIN {X 0,Y 439.792,Z 155.811,A -85,B 0,C 180,E1 -9255.858,E2 -9255.858} C_VEL
LIN {X 0,Y 441.982,Z 169.392,A -85,B 0,C 180,E1 -9256.153,E2 -9256.153} C_VEL
LIN {X 0,Y 441.594,Z 229.842,A -85,B 0,C 180,E1 -9257.155,E2 -9257.155} C_VEL
LIN {X 0,Y 441.403,Z 238.938,A -85,B 0,C 180,E1 -9257.412,E2 -9257.412} C_VEL
LIN {X 0,Y 441.322,Z 242.049,A -85,B 0,C 180,E1 -9257.519,E2 -9257.519} C_VEL
LIN {X 0,Y 440.573,Z 245.863,A -85,B 0,C 180,E1 -9257.646,E2 -9257.646} C_VEL
LIN {X 0,Y 437.589,Z 251.762,A -85,B 0,C 180,E1 -9257.847,E2 -9257.847} C_VEL
LIN {X 0,Y 434.58,Z 257.448,A -85,B 0,C 180,E1 -9258.119,E2 -9258.119} C_VEL
LIN {X 0,Y 433.789,Z 260.922,A -85,B 0,C 180,E1 -9258.354,E2 -9258.354} C_VEL
LIN {X 0,Y 433.267,Z 270.351,A -85,B 0,C 180,E1 -9259.131,E2 -9259.131} C_VEL
LIN {X 0,Y 432.935,Z 278.286,A -85,B 0,C 180,E1 -9259.95,E2 -9259.95} C_VEL
LIN {X 0,Y 432.572,Z 283.986,A -85,B 0,C 180,E1 -9260.649,E2 -9260.649} C_VEL
LIN {X 0,Y 432.183,Z 290.347,A -85,B 0,C 180,E1 -9261.584,E2 -9261.584} C_VEL
LIN {X 0,Y 431.961,Z 295.633,A -85,B 0,C 180,E1 -9262.521,E2 -9262.521} C_VEL
LIN {X 0,Y 431.821,Z 300.046,A -85,B 0,C 180,E1 -9263.458,E2 -9263.458} C_VEL
LIN {X 0,Y 431.48,Z 305.236,A -85,B 0,C 180,E1 -9264.86,E2 -9264.86} C_VEL
LIN {X 0,Y 431.38,Z 307.902,A -85,B 0,C 180,E1 -9265.795,E2 -9265.795} C_VEL
LIN {X 0,Y 431.306,Z 310.819,A -85,B 0,C 180,E1 -9267.198,E2 -9267.198} C_VEL
LIN {X 0,Y 431.206,Z 312.098,A -85,B 0,C 180,E1 -9268.132,E2 -9268.132} C_VEL
LIN {X 0,Y 431.148,Z 312.907,A -85,B 0,C 180,E1 -9269.066,E2 -9269.066} C_VEL
LIN {X 0,Y 431.144,Z 313.214,A -85,B 0,C 180,E1 -9270,E2 -9270} C_VEL
LIN {X 0,Y 431.148,Z 312.939,A -85,B 0,C 180,E1 -9270.934,E2 -9270.934} C_VEL
LIN {X 0,Y 431.206,Z 312.197,A -85,B 0,C 180,E1 -9271.868,E2 -9271.868} C_VEL
LIN {X 0,Y 431.304,Z 310.985,A -85,B 0,C 180,E1 -9272.802,E2 -9272.802} C_VEL
LIN {X 0,Y 431.369,Z 308.137,A -85,B 0,C 180,E1 -9274.204,E2 -9274.204} C_VEL
LIN {X 0,Y 431.474,Z 305.545,A -85,B 0,C 180,E1 -9275.14,E2 -9275.14} C_VEL
LIN {X 0,Y 431.781,Z 300.438,A -85,B 0,C 180,E1 -9276.542,E2 -9276.542} C_VEL
LIN {X 0,Y 431.959,Z 294.947,A -85,B 0,C 180,E1 -9277.714,E2 -9277.714} C_VEL
LIN {X 0,Y 432.358,Z 288.049,A -85,B 0,C 180,E1 -9278.883,E2 -9278.883} C_VEL
LIN {X 0,Y 432.819,Z 280.127,A -85,B 0,C 180,E1 -9279.934,E2 -9279.934} C_VEL
LIN {X 0,Y 433.188,Z 272.572,A -85,B 0,C 180,E1 -9280.753,E2 -9280.753} C_VEL
LIN {X 0,Y 433.554,Z 264.655,A -85,B 0,C 180,E1 -9281.453,E2 -9281.453} C_VEL
LIN {X 0,Y 433.96,Z 256.481,A -85,B 0,C 180,E1 -9282.035,E2 -9282.035} C_VEL
LIN {X 0,Y 434.268,Z 248.205,A -85,B 0,C 180,E1 -9282.501,E2 -9282.501} C_VEL
LIN {X 0,Y 434.553,Z 239.273,A -85,B 0,C 180,E1 -9282.878,E2 -9282.878} C_VEL
LIN {X 0,Y 434.76,Z 230.556,A -85,B 0,C 180,E1 -9283.133,E2 -9283.133} C_VEL
LIN {X 0,Y 435.052,Z 169.347,A -85,B 0,C 180,E1 -9284.172,E2 -9284.172} C_VEL
LIN {X 0,Y 432.553,Z 154.521,A -85,B 0,C 180,E1 -9284.526,E2 -9284.526} C_VEL
LIN {X 0,Y 432.501,Z 153.329,A -85,B 0,C 180,E1 -9284.708,E2 -9284.708} C_VEL
LIN {X 0,Y 433.009,Z 140.377,A -85,B 0,C 180,E1 -9287.961,E2 -9287.961} C_VEL
LIN {X 0,Y 433.057,Z 133.506,A -85,B 0,C 180,E1 -9289.733,E2 -9289.733} C_VEL
LIN {X 0,Y 432.445,Z 129.551,A -85,B 0,C 180,E1 -9290.824,E2 -9290.824} C_VEL
LIN {X 0,Y 432.38,Z 129.442,A -85,B 0,C 180,E1 -9294.462,E2 -9294.462} C_VEL
LIN {X 0,Y 432.391,Z 129.434,A -85,B 0,C 180,E1 -9297.071,E2 -9297.071} C_VEL
LIN {X 0,Y 432.348,Z 129.443,A -85,B 0,C 180,E1 -9300.51,E2 -9300.51} C_VEL
LIN {X 0,Y 432.359,Z 129.443,A -85,B 0,C 180,E1 -9304.003,E2 -9304.003} C_VEL
LIN {X 0,Y 432.328,Z 129.441,A -85,B 0,C 180,E1 -9307.198,E2 -9307.198} C_VEL
LIN {X 0,Y 432.341,Z 129.443,A -85,B 0,C 180,E1 -9310.18,E2 -9310.18} C_VEL
LIN {X 0,Y 432.316,Z 129.443,A -85,B 0,C 180,E1 -9313.061,E2 -9313.061} C_VEL
LIN {X 0,Y 432.332,Z 129.448,A -85,B 0,C 180,E1 -9315.664,E2 -9315.664} C_VEL
LIN {X 0,Y 432.331,Z 129.441,A -85,B 0,C 180,E1 -9318.398,E2 -9318.398} C_VEL
LIN {X 0,Y 432.334,Z 129.443,A -85,B 0,C 180,E1 -9321.85,E2 -9321.85} C_VEL
LIN {X 0,Y 432.34,Z 129.447,A -85,B 0,C 180,E1 -9325.323,E2 -9325.323} C_VEL
LIN {X 0,Y 432.32,Z 129.444,A -85,B 0,C 180,E1 -9328.654,E2 -9328.654} C_VEL
LIN {X 0,Y 432.38,Z 129.435,A -85,B 0,C 180,E1 -9331.876,E2 -9331.876} C_VEL
LIN {X 0,Y 432.35,Z 129.445,A -85,B 0,C 180,E1 -9334.999,E2 -9334.999} C_VEL
LIN {X 0,Y 432.356,Z 129.438,A -85,B 0,C 180,E1 -9338.046,E2 -9338.046} C_VEL
LIN {X 0,Y 432.385,Z 129.437,A -85,B 0,C 180,E1 -9341.029,E2 -9341.029} C_VEL
LIN {X 0,Y 432.429,Z 129.429,A -85,B 0,C 180,E1 -9343.961,E2 -9343.961} C_VEL
LIN {X 0,Y 432.479,Z 129.423,A -85,B 0,C 180,E1 -9347.804,E2 -9347.804} C_VEL
LIN {X 0,Y 432.491,Z 129.421,A -85,B 0,C 180,E1 -9351.59,E2 -9351.59} C_VEL
LIN {X 0,Y 432.596,Z 129.412,A -85,B 0,C 180,E1 -9354.406,E2 -9354.406} C_VEL
LIN {X 0,Y 432.604,Z 129.413,A -85,B 0,C 180,E1 -9358.138,E2 -9358.138} C_VEL
LIN {X 0,Y 432.732,Z 129.398,A -85,B 0,C 180,E1 -9360,E2 -9360} C_VEL
LIN {X 0,Y 432.591,Z 129.408,A -85,B 0,C 180,E1 -9362.794,E2 -9362.794} C_VEL
LIN {X 0,Y 432.571,Z 129.411,A -85,B 0,C 180,E1 -9366.53,E2 -9366.53} C_VEL
LIN {X 0,Y 432.441,Z 129.431,A -85,B 0,C 180,E1 -9369.353,E2 -9369.353} C_VEL
LIN {X 0,Y 432.429,Z 129.429,A -85,B 0,C 180,E1 -9372.803,E2 -9372.803} C_VEL
LIN {X 0,Y 432.411,Z 129.431,A -85,B 0,C 180,E1 -9376.479,E2 -9376.479} C_VEL
LIN {X 0,Y 432.337,Z 129.44,A -85,B 0,C 180,E1 -9379.96,E2 -9379.96} C_VEL
LIN {X 0,Y 432.317,Z 129.448,A -85,B 0,C 180,E1 -9382.964,E2 -9382.964} C_VEL
LIN {X 0,Y 432.362,Z 129.437,A -85,B 0,C 180,E1 -9386.032,E2 -9386.032} C_VEL
LIN {X 0,Y 432.341,Z 129.443,A -85,B 0,C 180,E1 -9389.187,E2 -9389.187} C_VEL
LIN {X 0,Y 432.321,Z 129.446,A -85,B 0,C 180,E1 -9392.443,E2 -9392.443} C_VEL
LIN {X 0,Y 432.343,Z 129.439,A -85,B 0,C 180,E1 -9395.632,E2 -9395.632} C_VEL
LIN {X 0,Y 432.336,Z 129.444,A -85,B 0,C 180,E1 -9398.714,E2 -9398.714} C_VEL
LIN {X 0,Y 432.331,Z 129.442,A -85,B 0,C 180,E1 -9401.797,E2 -9401.797} C_VEL
LIN {X 0,Y 432.331,Z 129.447,A -85,B 0,C 180,E1 -9404.347,E2 -9404.347} C_VEL
LIN {X 0,Y 432.318,Z 129.442,A -85,B 0,C 180,E1 -9407.016,E2 -9407.016} C_VEL
LIN {X 0,Y 432.331,Z 129.445,A -85,B 0,C 180,E1 -9409.821,E2 -9409.821} C_VEL
LIN {X 0,Y 432.306,Z 129.444,A -85,B 0,C 180,E1 -9413.022,E2 -9413.022} C_VEL
LIN {X 0,Y 432.358,Z 129.442,A -85,B 0,C 180,E1 -9415.997,E2 -9415.997} C_VEL
LIN {X 0,Y 432.346,Z 129.443,A -85,B 0,C 180,E1 -9419.49,E2 -9419.49} C_VEL
LIN {X 0,Y 432.39,Z 129.434,A -85,B 0,C 180,E1 -9422.928,E2 -9422.928} C_VEL
LIN {X 0,Y 432.435,Z 129.59,A -85,B 0,C 180,E1 -9426.282,E2 -9426.282} C_VEL
LIN {X 0,Y 433.72,Z 137.933,A -85,B 0,C 180,E1 -9428.368,E2 -9428.368} C_VEL
LIN {X 0,Y 433.372,Z 147.46,A -85,B 0,C 180,E1 -9430.598,E2 -9430.598} C_VEL
LIN {X 0,Y 432.598,Z 163.124,A -85,B 0,C 180,E1 -9434.21,E2 -9434.21} C_VEL
LIN {X 0,Y 432.373,Z 168.795,A -85,B 0,C 180,E1 -9435.468,E2 -9435.468} C_VEL
LIN {X 0,Y 432.755,Z 171.996,A -85,B 0,C 180,E1 -9435.586,E2 -9435.586} C_VEL
LIN {X 0,Y 434.891,Z 187.592,A -85,B 0,C 180,E1 -9435.918,E2 -9435.918} C_VEL
LIN {X 0,Y 434.666,Z 244.818,A -85,B 0,C 180,E1 -9436.885,E2 -9436.885} C_VEL
LIN {X 0,Y 434.347,Z 254.17,A -85,B 0,C 180,E1 -9437.145,E2 -9437.145} C_VEL
LIN {X 0,Y 434.019,Z 263.835,A -85,B 0,C 180,E1 -9437.551,E2 -9437.551} C_VEL
LIN {X 0,Y 433.645,Z 272.998,A -85,B 0,C 180,E1 -9438.075,E2 -9438.075} C_VEL
LIN {X 0,Y 433.156,Z 283.805,A -85,B 0,C 180,E1 -9438.891,E2 -9438.891} C_VEL
LIN {X 0,Y 432.626,Z 293.114,A -85,B 0,C 180,E1 -9439.825,E2 -9439.825} C_VEL
LIN {X 0,Y 432.322,Z 299.787,A -85,B 0,C 180,E1 -9440.645,E2 -9440.645} C_VEL
LIN {X 0,Y 431.963,Z 306.12,A -85,B 0,C 180,E1 -9441.58,E2 -9441.58} C_VEL
LIN {X 0,Y 431.73,Z 311.384,A -85,B 0,C 180,E1 -9442.517,E2 -9442.517} C_VEL
LIN {X 0,Y 431.521,Z 315.772,A -85,B 0,C 180,E1 -9443.454,E2 -9443.454} C_VEL
LIN {X 0,Y 431.394,Z 319.425,A -85,B 0,C 180,E1 -9444.391,E2 -9444.391} C_VEL
LIN {X 0,Y 431.303,Z 322.422,A -85,B 0,C 180,E1 -9445.327,E2 -9445.327} C_VEL
LIN {X 0,Y 431.22,Z 324.746,A -85,B 0,C 180,E1 -9446.262,E2 -9446.262} C_VEL
LIN {X 0,Y 431.207,Z 326.493,A -85,B 0,C 180,E1 -9447.198,E2 -9447.198} C_VEL
LIN {X 0,Y 431.197,Z 327.745,A -85,B 0,C 180,E1 -9448.132,E2 -9448.132} C_VEL
LIN {X 0,Y 431.146,Z 328.523,A -85,B 0,C 180,E1 -9449.066,E2 -9449.066} C_VEL
LIN {X 0,Y 431.142,Z 328.817,A -85,B 0,C 180,E1 -9450,E2 -9450} C_VEL
LIN {X 0,Y 431.146,Z 328.521,A -85,B 0,C 180,E1 -9450.934,E2 -9450.934} C_VEL
LIN {X 0,Y 431.197,Z 327.739,A -85,B 0,C 180,E1 -9451.868,E2 -9451.868} C_VEL
LIN {X 0,Y 431.207,Z 326.483,A -85,B 0,C 180,E1 -9452.803,E2 -9452.803} C_VEL
LIN {X 0,Y 431.242,Z 323.577,A -85,B 0,C 180,E1 -9454.206,E2 -9454.206} C_VEL
LIN {X 0,Y 431.365,Z 320.93,A -85,B 0,C 180,E1 -9455.141,E2 -9455.141} C_VEL
LIN {X 0,Y 431.453,Z 317.202,A -85,B 0,C 180,E1 -9456.191,E2 -9456.191} C_VEL
LIN {X 0,Y 431.627,Z 312.526,A -85,B 0,C 180,E1 -9457.25,E2 -9457.25} C_VEL
LIN {X 0,Y 431.84,Z 307.503,A -85,B 0,C 180,E1 -9458.187,E2 -9458.187} C_VEL
LIN {X 0,Y 432.209,Z 301.455,A -85,B 0,C 180,E1 -9459.122,E2 -9459.122} C_VEL
LIN {X 0,Y 432.586,Z 294.093,A -85,B 0,C 180,E1 -9460.058,E2 -9460.058} C_VEL
LIN {X 0,Y 433.042,Z 286.211,A -85,B 0,C 180,E1 -9460.875,E2 -9460.875} C_VEL
LIN {X 0,Y 433.442,Z 277.881,A -85,B 0,C 180,E1 -9461.575,E2 -9461.575} C_VEL
LIN {X 0,Y 433.925,Z 267.243,A -85,B 0,C 180,E1 -9462.274,E2 -9462.274} C_VEL
LIN {X 0,Y 434.273,Z 255.666,A -85,B 0,C 180,E1 -9462.798,E2 -9462.798} C_VEL
LIN {X 0,Y 434.571,Z 245.977,A -85,B 0,C 180,E1 -9463.086,E2 -9463.086} C_VEL
LIN {X 0,Y 435.019,Z 188.989,A -85,B 0,C 180,E1 -9464.049,E2 -9464.049} C_VEL
LIN {X 0,Y 432.776,Z 171.998,A -85,B 0,C 180,E1 -9464.407,E2 -9464.407} C_VEL
LIN {X 0,Y 432.392,Z 168.904,A -85,B 0,C 180,E1 -9464.514,E2 -9464.514} C_VEL
LIN {X 0,Y 432.913,Z 155.759,A -85,B 0,C 180,E1 -9467.478,E2 -9467.478} C_VEL
LIN {X 0,Y 433.614,Z 142.115,A -85,B 0,C 180,E1 -9470.642,E2 -9470.642} C_VEL
LIN {X 0,Y 433.656,Z 136.847,A -85,B 0,C 180,E1 -9471.885,E2 -9471.885} C_VEL
LIN {X 0,Y 432.436,Z 129.565,A -85,B 0,C 180,E1 -9473.718,E2 -9473.718} C_VEL
LIN {X 0,Y 432.392,Z 129.434,A -85,B 0,C 180,E1 -9477.072,E2 -9477.072} C_VEL
LIN {X 0,Y 432.348,Z 129.443,A -85,B 0,C 180,E1 -9480.511,E2 -9480.511} C_VEL
LIN {X 0,Y 432.36,Z 129.442,A -85,B 0,C 180,E1 -9484.004,E2 -9484.004} C_VEL
LIN {X 0,Y 432.323,Z 129.442,A -85,B 0,C 180,E1 -9487.197,E2 -9487.197} C_VEL
LIN {X 0,Y 432.334,Z 129.445,A -85,B 0,C 180,E1 -9490.179,E2 -9490.179} C_VEL
LIN {X 0,Y 432.317,Z 129.443,A -85,B 0,C 180,E1 -9493.061,E2 -9493.061} C_VEL
LIN {X 0,Y 432.333,Z 129.447,A -85,B 0,C 180,E1 -9495.665,E2 -9495.665} C_VEL
LIN {X 0,Y 432.333,Z 129.441,A -85,B 0,C 180,E1 -9498.398,E2 -9498.398} C_VEL
LIN {X 0,Y 432.336,Z 129.443,A -85,B 0,C 180,E1 -9501.85,E2 -9501.85} C_VEL
LIN {X 0,Y 432.342,Z 129.446,A -85,B 0,C 180,E1 -9505.323,E2 -9505.323} C_VEL
LIN {X 0,Y 432.322,Z 129.443,A -85,B 0,C 180,E1 -9508.654,E2 -9508.654} C_VEL
LIN {X 0,Y 432.383,Z 129.435,A -85,B 0,C 180,E1 -9511.877,E2 -9511.877} C_VEL
LIN {X 0,Y 432.353,Z 129.445,A -85,B 0,C 180,E1 -9514.999,E2 -9514.999} C_VEL
LIN {X 0,Y 432.359,Z 129.437,A -85,B 0,C 180,E1 -9518.046,E2 -9518.046} C_VEL
LIN {X 0,Y 432.388,Z 129.438,A -85,B 0,C 180,E1 -9521.03,E2 -9521.03} C_VEL
LIN {X 0,Y 432.432,Z 129.428,A -85,B 0,C 180,E1 -9523.961,E2 -9523.961} C_VEL
LIN {X 0,Y 432.461,Z 129.425,A -85,B 0,C 180,E1 -9527.804,E2 -9527.804} C_VEL
LIN {X 0,Y 432.494,Z 129.421,A -85,B 0,C 180,E1 -9531.59,E2 -9531.59} C_VEL
LIN {X 0,Y 432.596,Z 129.413,A -85,B 0,C 180,E1 -9534.406,E2 -9534.406} C_VEL
LIN {X 0,Y 432.605,Z 129.414,A -85,B 0,C 180,E1 -9538.138,E2 -9538.138} C_VEL
LIN {X 0,Y 432.734,Z 129.397,A -85,B 0,C 180,E1 -9540,E2 -9540} C_VEL
LIN {X 0,Y 432.593,Z 129.408,A -85,B 0,C 180,E1 -9542.794,E2 -9542.794} C_VEL
LIN {X 0,Y 432.574,Z 129.411,A -85,B 0,C 180,E1 -9546.53,E2 -9546.53} C_VEL
LIN {X 0,Y 432.446,Z 129.429,A -85,B 0,C 180,E1 -9549.353,E2 -9549.353} C_VEL
LIN {X 0,Y 432.447,Z 129.426,A -85,B 0,C 180,E1 -9552.812,E2 -9552.812} C_VEL
LIN {X 0,Y 432.414,Z 129.43,A -85,B 0,C 180,E1 -9556.479,E2 -9556.479} C_VEL
LIN {X 0,Y 432.34,Z 129.44,A -85,B 0,C 180,E1 -9559.96,E2 -9559.96} C_VEL
LIN {X 0,Y 432.32,Z 129.446,A -85,B 0,C 180,E1 -9562.964,E2 -9562.964} C_VEL
LIN {X 0,Y 432.366,Z 129.436,A -85,B 0,C 180,E1 -9566.032,E2 -9566.032} C_VEL
LIN {X 0,Y 432.345,Z 129.443,A -85,B 0,C 180,E1 -9569.187,E2 -9569.187} C_VEL
LIN {X 0,Y 432.325,Z 129.444,A -85,B 0,C 180,E1 -9572.443,E2 -9572.443} C_VEL
LIN {X 0,Y 432.347,Z 129.439,A -85,B 0,C 180,E1 -9575.632,E2 -9575.632} C_VEL
LIN {X 0,Y 432.34,Z 129.446,A -85,B 0,C 180,E1 -9578.714,E2 -9578.714} C_VEL
LIN {X 0,Y 432.334,Z 129.441,A -85,B 0,C 180,E1 -9581.797,E2 -9581.797} C_VEL
LIN {X 0,Y 432.335,Z 129.447,A -85,B 0,C 180,E1 -9584.347,E2 -9584.347} C_VEL
LIN {X 0,Y 432.322,Z 129.442,A -85,B 0,C 180,E1 -9587.016,E2 -9587.016} C_VEL
LIN {X 0,Y 432.343,Z 129.442,A -85,B 0,C 180,E1 -9589.82,E2 -9589.82} C_VEL
LIN {X 0,Y 432.317,Z 129.442,A -85,B 0,C 180,E1 -9593.023,E2 -9593.023} C_VEL
LIN {X 0,Y 432.361,Z 129.444,A -85,B 0,C 180,E1 -9595.996,E2 -9595.996} C_VEL
LIN {X 0,Y 432.349,Z 129.441,A -85,B 0,C 180,E1 -9599.49,E2 -9599.49} C_VEL
LIN {X 0,Y 432.392,Z 129.433,A -85,B 0,C 180,E1 -9602.928,E2 -9602.928} C_VEL
LIN {X 0,Y 432.37,Z 129.441,A -85,B 0,C 180,E1 -9606.023,E2 -9606.023} C_VEL
LIN {X 0,Y 432.427,Z 129.618,A -85,B 0,C 180,E1 -9609.299,E2 -9609.299} C_VEL
LIN {X 0,Y 433.155,Z 134.691,A -85,B 0,C 180,E1 -9610.677,E2 -9610.677} C_VEL
LIN {X 0,Y 432.783,Z 145.785,A -85,B 0,C 180,E1 -9613.504,E2 -9613.504} C_VEL
LIN {X 0,Y 432.507,Z 154.182,A -85,B 0,C 180,E1 -9615.541,E2 -9615.541} C_VEL
LIN {X 0,Y 432.964,Z 157.01,A -85,B 0,C 180,E1 -9615.648,E2 -9615.648} C_VEL
LIN {X 0,Y 435.039,Z 169.549,A -85,B 0,C 180,E1 -9615.928,E2 -9615.928} C_VEL
LIN {X 0,Y 434.691,Z 229.989,A -85,B 0,C 180,E1 -9616.947,E2 -9616.947} C_VEL
LIN {X 0,Y 434.482,Z 239.079,A -85,B 0,C 180,E1 -9617.208,E2 -9617.208} C_VEL
LIN {X 0,Y 434.236,Z 248.667,A -85,B 0,C 180,E1 -9617.617,E2 -9617.617} C_VEL
LIN {X 0,Y 433.858,Z 258.707,A -85,B 0,C 180,E1 -9618.199,E2 -9618.199} C_VEL
LIN {X 0,Y 433.789,Z 260.922,A -85,B 0,C 180,E1 -9618.354,E2 -9618.354} C_VEL
LIN {X 0,Y 432.953,Z 266.199,A -85,B 0,C 180,E1 -9618.746,E2 -9618.746} C_VEL
LIN {X 0,Y 429.723,Z 274.189,A -85,B 0,C 180,E1 -9619.406,E2 -9619.406} C_VEL
LIN {X 0,Y 426.43,Z 281.546,A -85,B 0,C 180,E1 -9620.165,E2 -9620.165} C_VEL
LIN {X 0,Y 425.466,Z 285.604,A -85,B 0,C 180,E1 -9620.702,E2 -9620.702} C_VEL
LIN {X 0,Y 425.07,Z 291.892,A -85,B 0,C 180,E1 -9621.682,E2 -9621.682} C_VEL
LIN {X 0,Y 424.816,Z 298.105,A -85,B 0,C 180,E1 -9622.873,E2 -9622.873} C_VEL
LIN {X 0,Y 424.534,Z 303.853,A -85,B 0,C 180,E1 -9624.299,E2 -9624.299} C_VEL
LIN {X 0,Y 424.331,Z 306.854,A -85,B 0,C 180,E1 -9625.25,E2 -9625.25} C_VEL
LIN {X 0,Y 424.265,Z 309.178,A -85,B 0,C 180,E1 -9626.201,E2 -9626.201} C_VEL
LIN {X 0,Y 424.224,Z 310.948,A -85,B 0,C 180,E1 -9627.151,E2 -9627.151} C_VEL
LIN {X 0,Y 424.134,Z 312.226,A -85,B 0,C 180,E1 -9628.101,E2 -9628.101} C_VEL
LIN {X 0,Y 424.069,Z 313.035,A -85,B 0,C 180,E1 -9629.05,E2 -9629.05} C_VEL
LIN {X 0,Y 424.062,Z 313.342,A -85,B 0,C 180,E1 -9630,E2 -9630} C_VEL
LIN {X 0,Y 424.069,Z 313.067,A -85,B 0,C 180,E1 -9630.949,E2 -9630.949} C_VEL
LIN {X 0,Y 424.134,Z 312.324,A -85,B 0,C 180,E1 -9631.899,E2 -9631.899} C_VEL
LIN {X 0,Y 424.222,Z 311.113,A -85,B 0,C 180,E1 -9632.849,E2 -9632.849} C_VEL
LIN {X 0,Y 424.281,Z 308.265,A -85,B 0,C 180,E1 -9634.275,E2 -9634.275} C_VEL
LIN {X 0,Y 424.417,Z 305.672,A -85,B 0,C 180,E1 -9635.225,E2 -9635.225} C_VEL
LIN {X 0,Y 424.717,Z 300.565,A -85,B 0,C 180,E1 -9636.651,E2 -9636.651} C_VEL
LIN {X 0,Y 424.912,Z 295.073,A -85,B 0,C 180,E1 -9637.842,E2 -9637.842} C_VEL
LIN {X 0,Y 425.339,Z 288.175,A -85,B 0,C 180,E1 -9639.031,E2 -9639.031} C_VEL
LIN {X 0,Y 425.826,Z 280.251,A -85,B 0,C 180,E1 -9640.099,E2 -9640.099} C_VEL
LIN {X 0,Y 426.221,Z 272.696,A -85,B 0,C 180,E1 -9640.931,E2 -9640.931} C_VEL
LIN {X 0,Y 426.62,Z 264.778,A -85,B 0,C 180,E1 -9641.642,E2 -9641.642} C_VEL
LIN {X 0,Y 427.005,Z 256.603,A -85,B 0,C 180,E1 -9642.234,E2 -9642.234} C_VEL
LIN {X 0,Y 427.341,Z 248.324,A -85,B 0,C 180,E1 -9642.707,E2 -9642.707} C_VEL
LIN {X 0,Y 427.659,Z 239.389,A -85,B 0,C 180,E1 -9643.089,E2 -9643.089} C_VEL
LIN {X 0,Y 427.848,Z 230.025,A -85,B 0,C 180,E1 -9643.364,E2 -9643.364} C_VEL
LIN {X 0,Y 428.109,Z 169.617,A -85,B 0,C 180,E1 -9644.404,E2 -9644.404} C_VEL
LIN {X 0,Y 425.551,Z 154.635,A -85,B 0,C 180,E1 -9644.77,E2 -9644.77} C_VEL
LIN {X 0,Y 425.485,Z 153.449,A -85,B 0,C 180,E1 -9644.956,E2 -9644.956} C_VEL
LIN {X 0,Y 426.037,Z 140.469,A -85,B 0,C 180,E1 -9648.266,E2 -9648.266} C_VEL
LIN {X 0,Y 426.006,Z 134.287,A -85,B 0,C 180,E1 -9649.889,E2 -9649.889} C_VEL
LIN {X 0,Y 425.382,Z 130.416,A -85,B 0,C 180,E1 -9650.996,E2 -9650.996} C_VEL
LIN {X 0,Y 425.322,Z 130.319,A -85,B 0,C 180,E1 -9654.657,E2 -9654.657} C_VEL
LIN {X 0,Y 425.349,Z 130.311,A -85,B 0,C 180,E1 -9657.557,E2 -9657.557} C_VEL
LIN {X 0,Y 425.288,Z 130.319,A -85,B 0,C 180,E1 -9660.816,E2 -9660.816} C_VEL
LIN {X 0,Y 425.311,Z 130.32,A -85,B 0,C 180,E1 -9664.288,E2 -9664.288} C_VEL
LIN {X 0,Y 425.284,Z 130.322,A -85,B 0,C 180,E1 -9667.693,E2 -9667.693} C_VEL
LIN {X 0,Y 425.283,Z 130.319,A -85,B 0,C 180,E1 -9670.521,E2 -9670.521} C_VEL
LIN {X 0,Y 425.257,Z 130.324,A -85,B 0,C 180,E1 -9673.351,E2 -9673.351} C_VEL
LIN {X 0,Y 425.256,Z 130.322,A -85,B 0,C 180,E1 -9676.649,E2 -9676.649} C_VEL
LIN {X 0,Y 425.284,Z 130.321,A -85,B 0,C 180,E1 -9679.872,E2 -9679.872} C_VEL
LIN {X 0,Y 425.277,Z 130.319,A -85,B 0,C 180,E1 -9682.488,E2 -9682.488} C_VEL
LIN {X 0,Y 425.307,Z 130.317,A -85,B 0,C 180,E1 -9685.817,E2 -9685.817} C_VEL
LIN {X 0,Y 425.289,Z 130.324,A -85,B 0,C 180,E1 -9689.239,E2 -9689.239} C_VEL
LIN {X 0,Y 425.347,Z 130.312,A -85,B 0,C 180,E1 -9692.442,E2 -9692.442} C_VEL
LIN {X 0,Y 425.35,Z 130.311,A -85,B 0,C 180,E1 -9695.602,E2 -9695.602} C_VEL
LIN {X 0,Y 425.292,Z 130.323,A -85,B 0,C 180,E1 -9698.681,E2 -9698.681} C_VEL
LIN {X 0,Y 425.332,Z 130.312,A -85,B 0,C 180,E1 -9701.703,E2 -9701.703} C_VEL
LIN {X 0,Y 425.347,Z 130.316,A -85,B 0,C 180,E1 -9704.671,E2 -9704.671} C_VEL
LIN {X 0,Y 425.429,Z 130.301,A -85,B 0,C 180,E1 -9707.599,E2 -9707.599} C_VEL
LIN {X 0,Y 425.441,Z 130.299,A -85,B 0,C 180,E1 -9711.45,E2 -9711.45} C_VEL
LIN {X 0,Y 425.553,Z 130.291,A -85,B 0,C 180,E1 -9714.313,E2 -9714.313} C_VEL
LIN {X 0,Y 425.574,Z 130.289,A -85,B 0,C 180,E1 -9718.107,E2 -9718.107} C_VEL
LIN {X 0,Y 425.702,Z 130.273,A -85,B 0,C 180,E1 -9720,E2 -9720} C_VEL
LIN {X 0,Y 425.545,Z 130.286,A -85,B 0,C 180,E1 -9722.84,E2 -9722.84} C_VEL
LIN {X 0,Y 425.572,Z 130.289,A -85,B 0,C 180,E1 -9725.686,E2 -9725.686} C_VEL
LIN {X 0,Y 425.441,Z 130.299,A -85,B 0,C 180,E1 -9728.55,E2 -9728.55} C_VEL
LIN {X 0,Y 425.41,Z 130.303,A -85,B 0,C 180,E1 -9732.402,E2 -9732.402} C_VEL
LIN {X 0,Y 425.387,Z 130.306,A -85,B 0,C 180,E1 -9736.312,E2 -9736.312} C_VEL
LIN {X 0,Y 425.327,Z 130.316,A -85,B 0,C 180,E1 -9739.636,E2 -9739.636} C_VEL
LIN {X 0,Y 425.305,Z 130.32,A -85,B 0,C 180,E1 -9743.365,E2 -9743.365} C_VEL
LIN {X 0,Y 425.345,Z 130.317,A -85,B 0,C 180,E1 -9746.844,E2 -9746.844} C_VEL
LIN {X 0,Y 425.289,Z 130.318,A -85,B 0,C 180,E1 -9749.72,E2 -9749.72} C_VEL
LIN {X 0,Y 425.28,Z 130.322,A -85,B 0,C 180,E1 -9753.048,E2 -9753.048} C_VEL
LIN {X 0,Y 425.281,Z 130.32,A -85,B 0,C 180,E1 -9755.929,E2 -9755.929} C_VEL
LIN {X 0,Y 425.279,Z 130.32,A -85,B 0,C 180,E1 -9759.041,E2 -9759.041} C_VEL
